//     IOTask Inputs/ControllerTags.CPX8_1[6,6] <-> Module 7 (CPX-AP-I-8DI-M8-3P)/Inputs/Input 5
//     IOTask Inputs/ControllerTags.CPX8_1[6,7] <-> Module 7 (CPX-AP-I-8DI-M8-3P)/Inputs/Input 6
//     IOTask Inputs/ControllerTags.CPX8_1[6,8] <-> Module 7 (CPX-AP-I-8DI-M8-3P)/Inputs/Input 7
//     IOTask Inputs/ControllerTags.CPX8_1[7,1] <-> Module 8 (CPX-AP-I-8DI-M8-3P)/Inputs/Input 0
//     IOTask Inputs/ControllerTags.CPX8_1[7,2] <-> Module 8 (CPX-AP-I-8DI-M8-3P)/Inputs/Input 1
//     IOTask Inputs/ControllerTags.CPX8_1[7,3] <-> Module 8 (CPX-AP-I-8DI-M8-3P)/Inputs/Input 2
//     IOTask Inputs/ControllerTags.CPX8_1[7,4] <-> Module 8 (CPX-AP-I-8DI-M8-3P)/Inputs/Input 3
//     IOTask Inputs/ControllerTags.CPX8_1[7,5] <-> Module 8 (CPX-AP-I-8DI-M8-3P)/Inputs/Input 4
//     IOTask Inputs/ControllerTags.CPX8_1[7,6] <-> Module 8 (CPX-AP-I-8DI-M8-3P)/Inputs/Input 5
//     IOTask Inputs/ControllerTags.CPX8_1[7,7] <-> Module 8 (CPX-AP-I-8DI-M8-3P)/Inputs/Input 6
//     IOTask Inputs/ControllerTags.CPX8_1[7,8] <-> Module 8 (CPX-AP-I-8DI-M8-3P)/Inputs/Input 7
//   PLC1/PLC1 Instance <-> Device 1 (EtherCAT)/Term 1 (EK1200)/Term 17 (EK1122)/Drive PA14401 (ASDA-A2-E CoE Drive)
//     PlcTask1 Inputs/ControllerTags.arErrorCodeDrive[44] <-> 1st Transmit PDO Mapping/Error code
//   PLC1/PLC1 Instance <-> Device 1 (EtherCAT)/Term 1 (EK1200)/Term 17 (EK1122)/Drive PA14501 (ASDA-A2-E CoE Drive)
//     PlcTask1 Inputs/ControllerTags.arErrorCodeDrive[45] <-> 1st Transmit PDO Mapping/Error code
//   PLC1/PLC1 Instance <-> Device 1 (EtherCAT)/Term 1 (EK1200)/Term 17 (EK1122)/Drive PA14601 (ASDA-A2-E CoE Drive)
//     PlcTask1 Inputs/ControllerTags.arErrorCodeDrive[46] <-> 1st TxPDO Mapping/Error code
//   PLC1/PLC1 Instance <-> Device 1 (EtherCAT)/Term 1 (EK1200)/Term 17 (EK1122)/Drive PA14701 (ASDA-A2-E CoE Drive)
//     PlcTask1 Inputs/ControllerTags.arErrorCodeDrive[47] <-> 1st Transmit PDO Mapping/Error code
//   PLC1/PLC1 Instance <-> Device 1 (EtherCAT)/Term 1 (EK1200)/Term 17 (EK1122)/WPI_1(WPI_EtherCAt_32Bits)
//     IOTask Outputs/ControllerTags.WPI_1[1,1] <-> DO Outputs/DataOutBit 1
//     IOTask Outputs/ControllerTags.WPI_1[1,2] <-> DO Outputs/DataOutBit  2
//     IOTask Outputs/ControllerTags.WPI_1[1,3] <-> DO Outputs/DataOutBit  3
//     IOTask Outputs/ControllerTags.WPI_1[1,4] <-> DO Outputs/DataOutBit  4
//     IOTask Outputs/ControllerTags.WPI_1[1,5] <-> DO Outputs/DataOutBit  5
//     IOTask Outputs/ControllerTags.WPI_1[1,6] <-> DO Outputs/DataOutBit  6
//     IOTask Outputs/ControllerTags.WPI_1[1,7] <-> DO Outputs/DataOutBit  7
//     IOTask Outputs/ControllerTags.WPI_1[1,8] <-> DO Outputs/DataOutBit  8
//     IOTask Outputs/ControllerTags.WPI_1[2,1] <-> DO Outputs/DataOutBit  9
//     IOTask Outputs/ControllerTags.WPI_1[2,2] <-> DO Outputs/DataOutBit  10
//     IOTask Outputs/ControllerTags.WPI_1[2,3] <-> DO Outputs/DataOutBit  11
//     IOTask Outputs/ControllerTags.WPI_1[2,4] <-> DO Outputs/DataOutBit  12
//     IOTask Outputs/ControllerTags.WPI_1[2,5] <-> DO Outputs/DataOutBit  13
//     IOTask Outputs/ControllerTags.WPI_1[2,6] <-> DO Outputs/DataOutBit  14
//     IOTask Outputs/ControllerTags.WPI_1[2,7] <-> DO Outputs/DataOutBit  15
//     IOTask Outputs/ControllerTags.WPI_1[2,8] <-> DO Outputs/DataOutBit  16
//     IOTask Outputs/ControllerTags.WPI_1[3,1] <-> DO Outputs/DataOutBit  17
//     IOTask Outputs/ControllerTags.WPI_1[3,2] <-> DO Outputs/DataOutBit  18
//     IOTask Outputs/ControllerTags.WPI_1[3,3] <-> DO Outputs/DataOutBit  19
//     IOTask Outputs/ControllerTags.WPI_1[3,4] <-> DO Outputs/DataOutBit  20
//     IOTask Outputs/ControllerTags.WPI_1[3,5] <-> DO Outputs/DataOutBit  21
//     IOTask Outputs/ControllerTags.WPI_1[3,6] <-> DO Outputs/DataOutBit  22
//     IOTask Outputs/ControllerTags.WPI_1[3,7] <-> DO Outputs/DataOutBit  23
//     IOTask Outputs/ControllerTags.WPI_1[3,8] <-> DO Outputs/DataOutBit  24
//     IOTask Outputs/ControllerTags.WPI_1[4,1] <-> DO Outputs/DataOutBit  25
//     IOTask Outputs/ControllerTags.WPI_1[4,2] <-> DO Outputs/DataOutBit  26
//     IOTask Outputs/ControllerTags.WPI_1[4,3] <-> DO Outputs/DataOutBit  27
//     IOTask Outputs/ControllerTags.WPI_1[4,4] <-> DO Outputs/DataOutBit  28
//     IOTask Outputs/ControllerTags.WPI_1[4,5] <-> DO Outputs/DataOutBit  29
//     IOTask Outputs/ControllerTags.WPI_1[4,6] <-> DO Outputs/DataOutBit  30
//     IOTask Outputs/ControllerTags.WPI_1[4,7] <-> DO Outputs/DataOutBit  31
//     IOTask Outputs/ControllerTags.WPI_1[4,8] <-> DO Outputs/DataOutBit  32
//   PLC1/PLC1 Instance <-> Device 1 (EtherCAT)/Term 1 (EK1200)/Term 17 (EK1122)/WPI_2(WPI_EtherCAt_32Bits)
//     IOTask Outputs/ControllerTags.WPI_2[1,1] <-> DO Outputs/DataOutBit 1
//     IOTask Outputs/ControllerTags.WPI_2[1,2] <-> DO Outputs/DataOutBit  2
//     IOTask Outputs/ControllerTags.WPI_2[1,3] <-> DO Outputs/DataOutBit  3
//     IOTask Outputs/ControllerTags.WPI_2[1,4] <-> DO Outputs/DataOutBit  4
//     IOTask Outputs/ControllerTags.WPI_2[1,5] <-> DO Outputs/DataOutBit  5
//     IOTask Outputs/ControllerTags.WPI_2[1,6] <-> DO Outputs/DataOutBit  6
//     IOTask Outputs/ControllerTags.WPI_2[1,7] <-> DO Outputs/DataOutBit  7
//     IOTask Outputs/ControllerTags.WPI_2[1,8] <-> DO Outputs/DataOutBit  8
//     IOTask Outputs/ControllerTags.WPI_2[2,1] <-> DO Outputs/DataOutBit  9
//     IOTask Outputs/ControllerTags.WPI_2[2,2] <-> DO Outputs/DataOutBit  10
//     IOTask Outputs/ControllerTags.WPI_2[2,3] <-> DO Outputs/DataOutBit  11
//     IOTask Outputs/ControllerTags.WPI_2[2,4] <-> DO Outputs/DataOutBit  12
//     IOTask Outputs/ControllerTags.WPI_2[2,5] <-> DO Outputs/DataOutBit  13
//     IOTask Outputs/ControllerTags.WPI_2[2,6] <-> DO Outputs/DataOutBit  14
//     IOTask Outputs/ControllerTags.WPI_2[2,7] <-> DO Outputs/DataOutBit  15
//     IOTask Outputs/ControllerTags.WPI_2[2,8] <-> DO Outputs/DataOutBit  16
//     IOTask Outputs/ControllerTags.WPI_2[3,1] <-> DO Outputs/DataOutBit  17
//     IOTask Outputs/ControllerTags.WPI_2[3,2] <-> DO Outputs/DataOutBit  18
//     IOTask Outputs/ControllerTags.WPI_2[3,3] <-> DO Outputs/DataOutBit  19
//     IOTask Outputs/ControllerTags.WPI_2[3,4] <-> DO Outputs/DataOutBit  20
//     IOTask Outputs/ControllerTags.WPI_2[3,5] <-> DO Outputs/DataOutBit  21
//     IOTask Outputs/ControllerTags.WPI_2[3,6] <-> DO Outputs/DataOutBit  22
//     IOTask Outputs/ControllerTags.WPI_2[3,7] <-> DO Outputs/DataOutBit  23
//     IOTask Outputs/ControllerTags.WPI_2[3,8] <-> DO Outputs/DataOutBit  24
//     IOTask Outputs/ControllerTags.WPI_2[4,1] <-> DO Outputs/DataOutBit  25
//     IOTask Outputs/ControllerTags.WPI_2[4,2] <-> DO Outputs/DataOutBit  26
//     IOTask Outputs/ControllerTags.WPI_2[4,3] <-> DO Outputs/DataOutBit  27
//     IOTask Outputs/ControllerTags.WPI_2[4,4] <-> DO Outputs/DataOutBit  28
//     IOTask Outputs/ControllerTags.WPI_2[4,5] <-> DO Outputs/DataOutBit  29
//     IOTask Outputs/ControllerTags.WPI_2[4,6] <-> DO Outputs/DataOutBit  30
//     IOTask Outputs/ControllerTags.WPI_2[4,7] <-> DO Outputs/DataOutBit  31
//     IOTask Outputs/ControllerTags.WPI_2[4,8] <-> DO Outputs/DataOutBit  32
//   PLC1/PLC1 Instance <-> Device 1 (EtherCAT)/Term 1 (EK1200)/Term 2 (EL1008)
//     IOTask Inputs/ControllerTags.EL1008[33,{1..8}] <-> Channel {1..8}/Input  (8 links)
//   PLC1/PLC1 Instance <-> Device 1 (EtherCAT)/Term 1 (EK1200)/Term 3 (EL1008)
//     IOTask Inputs/ControllerTags.EL1008[34,{1..8}] <-> Channel {1..8}/Input  (8 links)
//   PLC1/PLC1 Instance <-> Device 1 (EtherCAT)/Term 1 (EK1200)/Term 4 (EL1008)
//     IOTask Inputs/ControllerTags.EL1008[35,{1..8}] <-> Channel {1..8}/Input  (8 links)
//   PLC1/PLC1 Instance <-> Device 1 (EtherCAT)/Term 1 (EK1200)/Term 5 (EL1008)
//     IOTask Inputs/ControllerTags.EL1008[36,{1..8}] <-> Channel {1..8}/Input  (8 links)
//   PLC1/PLC1 Instance <-> Device 1 (EtherCAT)/Term 1 (EK1200)/Term 6 (EL1008)
//     IOTask Inputs/ControllerTags.EL1008[37,{1..8}] <-> Channel {1..8}/Input  (8 links)
//   PLC1/PLC1 Instance <-> Device 1 (EtherCAT)/Term 1 (EK1200)/Term 7 (EL2008)
//     IOTask Outputs/ControllerTags.EL2008[29,{1..8}] <-> Channel {1..8}/Output  (8 links)
//   PLC1/PLC1 Instance <-> Device 1 (EtherCAT)/Term 1 (EK1200)/Term 8 (EL2008)
//     IOTask Outputs/ControllerTags.EL2008[30,{1..8}] <-> Channel {1..8}/Output  (8 links)
//   PLC1/PLC1 Instance <-> Device 1 (EtherCAT)/Term 1 (EK1200)/Term 9 (EL2008)
//     IOTask Outputs/ControllerTags.EL2008[31,{1..8}] <-> Channel {1..8}/Output  (8 links)
//   PLC1/PLC1 Instance <-> Device 4 (EtherCAT)
//     CommunicationTask Inputs/EtherCatStates.Device2_nEcMasterDeviceId <-> InfoData/DevId
//     CommunicationTask Inputs/EtherCatStates.Device2_netID <-> InfoData/AmsNetId
//   PLC1/PLC1 Instance <-> Device 4 (EtherCAT)/Drive PA10101 (ASDA-A2-E CoE Drive)
//     PlcTask1 Inputs/ControllerTags.arErrorCodeDrive[1] <-> 1st TxPDO Mapping/Error code
//   PLC1/PLC1 Instance <-> Device 4 (EtherCAT)/Drive PA10201 (ASDA-A2-E CoE Drive)
//     PlcTask1 Inputs/ControllerTags.arErrorCodeDrive[2] <-> 1st TxPDO Mapping/Error code
//   PLC1/PLC1 Instance <-> Device 4 (EtherCAT)/Drive PA10301 (ASDA-A2-E CoE Drive)
//     PlcTask1 Inputs/ControllerTags.arErrorCodeDrive[3] <-> 1st TxPDO Mapping/Error code
//   PLC1/PLC1 Instance <-> Device 4 (EtherCAT)/Drive PA10401 (ASDA-A2-E CoE Drive)
//     PlcTask1 Inputs/ControllerTags.arErrorCodeDrive[4] <-> 1st TxPDO Mapping/Error code
//   PLC1/PLC1 Instance <-> Device 4 (EtherCAT)/Drive PA10501 (ASDA-A2-E CoE Drive)
//     PlcTask1 Inputs/ControllerTags.arErrorCodeDrive[5] <-> 1st TxPDO Mapping/Error code
//   PLC1/PLC1 Instance <-> Device 4 (EtherCAT)/Drive PA10601 (ASDA-A2-E CoE Drive)
//     PlcTask1 Inputs/ControllerTags.arErrorCodeDrive[6] <-> 1st TxPDO Mapping/Error code
//   PLC1/PLC1 Instance <-> Device 4 (EtherCAT)/Drive PA10701 (ASDA-A2-E CoE Drive)
//     PlcTask1 Inputs/ControllerTags.arErrorCodeDrive[7] <-> 1st TxPDO Mapping/Error code
//   PLC1/PLC1 Instance <-> Device 4 (EtherCAT)/Drive PA10801 (ASDA-A2-E CoE Drive)
//     PlcTask1 Inputs/ControllerTags.arErrorCodeDrive[8] <-> 1st TxPDO Mapping/Error code
//   PLC1/PLC1 Instance <-> Device 4 (EtherCAT)/Drive PA10901 (ASDA-A2-E CoE Drive)
//     PlcTask1 Inputs/ControllerTags.arErrorCodeDrive[9] <-> 1st TxPDO Mapping/Error code
//   PLC1/PLC1 Instance <-> Device 4 (EtherCAT)/Drive PA11001 (ASDA-A2-E CoE Drive)
//     PlcTask1 Inputs/ControllerTags.arErrorCodeDrive[10] <-> 1st TxPDO Mapping/Error code
//   PLC1/PLC1 Instance <-> Device 4 (EtherCAT)/Drive PA11101 (ASDA-A2-E CoE Drive)
//     PlcTask1 Inputs/ControllerTags.arErrorCodeDrive[11] <-> 1st TxPDO Mapping/Error code
//   PLC1/PLC1 Instance <-> Device 4 (EtherCAT)/Drive PA11201 (ASDA-A2-E CoE Drive)
//     PlcTask1 Inputs/ControllerTags.arErrorCodeDrive[12] <-> 1st TxPDO Mapping/Error code
//   PLC1/PLC1 Instance <-> Device 4 (EtherCAT)/Drive PA11301 (ASDA-A2-E CoE Drive)
//     PlcTask1 Inputs/ControllerTags.arErrorCodeDrive[13] <-> 1st TxPDO Mapping/Error code
//   PLC1/PLC1 Instance <-> Device 4 (EtherCAT)/Drive PA11401 (ASDA-A2-E CoE Drive)
//     PlcTask1 Inputs/ControllerTags.arErrorCodeDrive[14] <-> 1st TxPDO Mapping/Error code
//   PLC1/PLC1 Instance <-> Device 4 (EtherCAT)/Drive PA11501 (ASDA-A2-E CoE Drive)
//     PlcTask1 Inputs/ControllerTags.arErrorCodeDrive[15] <-> 1st TxPDO Mapping/Error code
//   PLC1/PLC1 Instance <-> Device 4 (EtherCAT)/Drive PA11601 (ASDA-A2-E CoE Drive)
//     PlcTask1 Inputs/ControllerTags.arErrorCodeDrive[16] <-> 1st TxPDO Mapping/Error code
//   PLC1/PLC1 Instance <-> Device 4 (EtherCAT)/Drive PA11701 (ASDA-A2-E CoE Drive)
//     PlcTask1 Inputs/ControllerTags.arErrorCodeDrive[17] <-> 1st TxPDO Mapping/Error code
//   PLC1/PLC1 Instance <-> Device 4 (EtherCAT)/Drive PA11801 (ASDA-A2-E CoE Drive)
//     PlcTask1 Inputs/ControllerTags.arErrorCodeDrive[18] <-> 1st TxPDO Mapping/Error code
//   PLC1/PLC1 Instance <-> Device 4 (EtherCAT)/Drive PA11901 (ASDA-A2-E CoE Drive)
//     PlcTask1 Inputs/ControllerTags.arErrorCodeDrive[19] <-> 1st TxPDO Mapping/Error code
//   PLC1/PLC1 Instance <-> Device 4 (EtherCAT)/Drive PA12001 (ASDA-A2-E CoE Drive)
//     PlcTask1 Inputs/ControllerTags.arErrorCodeDrive[20] <-> 1st TxPDO Mapping/Error code
//   PLC1/PLC1 Instance <-> Device 4 (EtherCAT)/Drive PA12101 (ASDA-A2-E CoE Drive)
//     PlcTask1 Inputs/ControllerTags.arErrorCodeDrive[41] <-> 1st TxPDO Mapping/Error code
//   PLC1/PLC1 Instance <-> Device 4 (EtherCAT)/Drive PA12201 (ASDA-A2-E CoE Drive)
//     PlcTask1 Inputs/ControllerTags.arErrorCodeDrive[21] <-> 1st TxPDO Mapping/Error code
//   PLC1/PLC1 Instance <-> Device 4 (EtherCAT)/Drive PA12301 (ASDA-A2-E CoE Drive)
//     PlcTask1 Inputs/ControllerTags.arErrorCodeDrive[22] <-> 1st TxPDO Mapping/Error code
//   PLC1/PLC1 Instance <-> Device 4 (EtherCAT)/Drive PA12401 (ASDA-A2-E CoE Drive)
//     PlcTask1 Inputs/ControllerTags.arErrorCodeDrive[23] <-> 1st TxPDO Mapping/Error code
//   PLC1/PLC1 Instance <-> Device 4 (EtherCAT)/Drive PA12501 (ASDA-A2-E CoE Drive)
//     PlcTask1 Inputs/ControllerTags.arErrorCodeDrive[24] <-> 1st TxPDO Mapping/Error code
//   PLC1/PLC1 Instance <-> Device 4 (EtherCAT)/Drive PA12601 (ASDA-A2-E CoE Drive)
//     PlcTask1 Inputs/ControllerTags.arErrorCodeDrive[25] <-> 1st TxPDO Mapping/Error code
//   PLC1/PLC1 Instance <-> Device 4 (EtherCAT)/Drive PA12701 (ASDA-A2-E CoE Drive)
//     PlcTask1 Inputs/ControllerTags.arErrorCodeDrive[26] <-> 1st TxPDO Mapping/Error code
//   PLC1/PLC1 Instance <-> Device 4 (EtherCAT)/Drive PA12801 (ASDA-A2-E CoE Drive)
//     PlcTask1 Inputs/ControllerTags.arErrorCodeDrive[27] <-> 1st TxPDO Mapping/Error code
//   PLC1/PLC1 Instance <-> Device 4 (EtherCAT)/Drive PA12901 (ASDA-A2-E CoE Drive)
//     PlcTask1 Inputs/ControllerTags.arErrorCodeDrive[28] <-> 1st TxPDO Mapping/Error code
//   PLC1/PLC1 Instance <-> Device 4 (EtherCAT)/Drive PA13001 (ASDA-A2-E CoE Drive)
//     PlcTask1 Inputs/ControllerTags.arErrorCodeDrive[29] <-> 1st TxPDO Mapping/Error code
//   PLC1/PLC1 Instance <-> Device 4 (EtherCAT)/Drive PA13101 (ASDA-A2-E CoE Drive)
//     PlcTask1 Inputs/ControllerTags.arErrorCodeDrive[30] <-> 1st TxPDO Mapping/Error code
//   PLC1/PLC1 Instance <-> Device 4 (EtherCAT)/Drive PA13201 (ASDA-A2-E CoE Drive)
//     PlcTask1 Inputs/ControllerTags.arErrorCodeDrive[42] <-> 1st TxPDO Mapping/Error code
//   PLC1/PLC1 Instance <-> Device 4 (EtherCAT)/Drive PA13301 (ASDA-A2-E CoE Drive)
//     PlcTask1 Inputs/ControllerTags.arErrorCodeDrive[31] <-> 1st Transmit PDO Mapping/Error code
//   PLC1/PLC1 Instance <-> Device 4 (EtherCAT)/Drive PA13401 (ASDA-A2-E CoE Drive)
//     PlcTask1 Inputs/ControllerTags.arErrorCodeDrive[32] <-> 1st Transmit PDO Mapping/Error code
//   PLC1/PLC1 Instance <-> Device 4 (EtherCAT)/Drive PA13501 (ASDA-A2-E CoE Drive)
//     PlcTask1 Inputs/ControllerTags.arErrorCodeDrive[33] <-> 1st Transmit PDO Mapping/Error code
//   PLC1/PLC1 Instance <-> Device 4 (EtherCAT)/Drive PA13601 (ASDA-A2-E CoE Drive)
//     PlcTask1 Inputs/ControllerTags.arErrorCodeDrive[34] <-> 1st TxPDO Mapping/Error code
//   PLC1/PLC1 Instance <-> Device 4 (EtherCAT)/Drive PA13701 (ASDA-A2-E CoE Drive)
//     PlcTask1 Inputs/ControllerTags.arErrorCodeDrive[35] <-> 1st TxPDO Mapping/Error code
//   PLC1/PLC1 Instance <-> Device 4 (EtherCAT)/Drive PA13801 (ASDA-A2-E CoE Drive)
//     PlcTask1 Inputs/ControllerTags.arErrorCodeDrive[36] <-> 1st TxPDO Mapping/Error code
//   PLC1/PLC1 Instance <-> Device 4 (EtherCAT)/Drive PA13901 (ASDA-A2-E CoE Drive)
//     PlcTask1 Inputs/ControllerTags.arErrorCodeDrive[37] <-> 1st TxPDO Mapping/Error code
//   PLC1/PLC1 Instance <-> Device 4 (EtherCAT)/Drive PA14001 (ASDA-A2-E CoE Drive)
//     PlcTask1 Inputs/ControllerTags.arErrorCodeDrive[38] <-> 1st TxPDO Mapping/Error code
//   PLC1/PLC1 Instance <-> Device 4 (EtherCAT)/Drive PA14101 (ASDA-A2-E CoE Drive)
//     PlcTask1 Inputs/ControllerTags.arErrorCodeDrive[39] <-> 1st TxPDO Mapping/Error code
//   PLC1/PLC1 Instance <-> Device 4 (EtherCAT)/Drive PA14201 (ASDA-A2-E CoE Drive)
//     PlcTask1 Inputs/ControllerTags.arErrorCodeDrive[40] <-> 1st TxPDO Mapping/Error code
//   PLC1/PLC1 Instance <-> Device 4 (EtherCAT)/Drive PA14301 (ASDA-A2-E CoE Drive)
//     PlcTask1 Inputs/ControllerTags.arErrorCodeDrive[43] <-> 1st TxPDO Mapping/Error code
//   PLC1/PLC1 Instance <-> Device 4 (EtherCAT)/Term CIM32101 (EK1100)/Term 110 (EL1008)
//     IOTask Inputs/ControllerTags.EL1008[1,{1..8}] <-> Channel {1..8}/Input  (8 links)
//   PLC1/PLC1 Instance <-> Device 4 (EtherCAT)/Term CIM32101 (EK1100)/Term 111 (EL1008)
//     IOTask Inputs/ControllerTags.EL1008[2,{1..8}] <-> Channel {1..8}/Input  (8 links)
//   PLC1/PLC1 Instance <-> Device 4 (EtherCAT)/Term CIM32101 (EK1100)/Term 112 (EL1008)
//     IOTask Inputs/ControllerTags.EL1008[3,{1..8}] <-> Channel {1..8}/Input  (8 links)
//   PLC1/PLC1 Instance <-> Device 4 (EtherCAT)/Term CIM32101 (EK1100)/Term 113 (EL1008)
//     IOTask Inputs/ControllerTags.EL1008[4,{1..8}] <-> Channel {1..8}/Input  (8 links)
//   PLC1/PLC1 Instance <-> Device 4 (EtherCAT)/Term CIM32101 (EK1100)/Term 114 (EL1008)
//     IOTask Inputs/ControllerTags.EL1008[5,{1..8}] <-> Channel {1..8}/Input  (8 links)
//   PLC1/PLC1 Instance <-> Device 4 (EtherCAT)/Term CIM32101 (EK1100)/Term 115 (EL1008)
//     IOTask Inputs/ControllerTags.EL1008[6,{1..8}] <-> Channel {1..8}/Input  (8 links)
//   PLC1/PLC1 Instance <-> Device 4 (EtherCAT)/Term CIM32101 (EK1100)/Term 116 (EL1008)
//     IOTask Inputs/ControllerTags.EL1008[7,{1..8}] <-> Channel {1..8}/Input  (8 links)
//   PLC1/PLC1 Instance <-> Device 4 (EtherCAT)/Term CIM32101 (EK1100)/Term 117 (EL1008)
//     IOTask Inputs/ControllerTags.EL1008[29,{1..8}] <-> Channel {1..8}/Input  (8 links)
//   PLC1/PLC1 Instance <-> Device 4 (EtherCAT)/Term CIM32101 (EK1100)/Term 118 (EL2008)
//     IOTask Outputs/ControllerTags.EL2008[1,{1..8}] <-> Channel {1..8}/Output  (8 links)
//   PLC1/PLC1 Instance <-> Device 4 (EtherCAT)/Term CIM32101 (EK1100)/Term 119 (EL2008)
//     IOTask Outputs/ControllerTags.EL2008[2,{1..8}] <-> Channel {1..8}/Output  (8 links)
//   PLC1/PLC1 Instance <-> Device 4 (EtherCAT)/Term CIM32101 (EK1100)/Term 120 (EL2008)
//     IOTask Outputs/ControllerTags.EL2008[3,{1..8}] <-> Channel {1..8}/Output  (8 links)
//   PLC1/PLC1 Instance <-> Device 4 (EtherCAT)/Term CIM32101 (EK1100)/Term 121 (EL2008)
//     IOTask Outputs/ControllerTags.EL2008[4,{1..8}] <-> Channel {1..8}/Output  (8 links)
//   PLC1/PLC1 Instance <-> Device 4 (EtherCAT)/Term CIM32101 (EK1100)/Term 122 (EL2008)
//     IOTask Outputs/ControllerTags.EL2008[5,{1..8}] <-> Channel {1..8}/Output  (8 links)
//   PLC1/PLC1 Instance <-> Device 4 (EtherCAT)/Term CIM32101 (EK1100)/Term 123 (EL2008)
//     IOTask Outputs/ControllerTags.EL2008[6,{1..8}] <-> Channel {1..8}/Output  (8 links)
//   PLC1/PLC1 Instance <-> Device 4 (EtherCAT)/Term CIM32101 (EK1100)/Term 124 (EL2008)
//     IOTask Outputs/ControllerTags.EL2008[7,{1..8}] <-> Channel {1..8}/Output  (8 links)
//   PLC1/PLC1 Instance <-> Device 4 (EtherCAT)/Term CIM33701 (EK1100)/Term 83 (EL1008)
//     IOTask Inputs/ControllerTags.EL1008[8,{1..8}] <-> Channel {1..8}/Input  (8 links)
//   PLC1/PLC1 Instance <-> Device 4 (EtherCAT)/Term CIM33701 (EK1100)/Term 84 (EL1008)
//     IOTask Inputs/ControllerTags.EL1008[9,{1..8}] <-> Channel {1..8}/Input  (8 links)
//   PLC1/PLC1 Instance <-> Device 4 (EtherCAT)/Term CIM33701 (EK1100)/Term 85 (EL1008)
//     IOTask Inputs/ControllerTags.EL1008[10,{1..8}] <-> Channel {1..8}/Input  (8 links)
//   PLC1/PLC1 Instance <-> Device 4 (EtherCAT)/Term CIM33701 (EK1100)/Term 86 (EL1008)
//     IOTask Inputs/ControllerTags.EL1008[11,{1..8}] <-> Channel {1..8}/Input  (8 links)
//   PLC1/PLC1 Instance <-> Device 4 (EtherCAT)/Term CIM33701 (EK1100)/Term 87 (EL1008)
//     IOTask Inputs/ControllerTags.EL1008[12,{1..8}] <-> Channel {1..8}/Input  (8 links)
//   PLC1/PLC1 Instance <-> Device 4 (EtherCAT)/Term CIM33701 (EK1100)/Term 88 (EL1008)
//     IOTask Inputs/ControllerTags.EL1008[13,{1..8}] <-> Channel {1..8}/Input  (8 links)
//   PLC1/PLC1 Instance <-> Device 4 (EtherCAT)/Term CIM33701 (EK1100)/Term 89 (EL1008)
//     IOTask Inputs/ControllerTags.EL1008[14,{1..8}] <-> Channel {1..8}/Input  (8 links)
//   PLC1/PLC1 Instance <-> Device 4 (EtherCAT)/Term CIM33701 (EK1100)/Term 90 (EL1008)
//     IOTask Inputs/ControllerTags.EL1008[30,{1..8}] <-> Channel {1..8}/Input  (8 links)
//   PLC1/PLC1 Instance <-> Device 4 (EtherCAT)/Term CIM33701 (EK1100)/Term 91 (EL2008)
//     IOTask Outputs/ControllerTags.EL2008[8,{1..8}] <-> Channel {1..8}/Output  (8 links)
//   PLC1/PLC1 Instance <-> Device 4 (EtherCAT)/Term CIM33701 (EK1100)/Term 92 (EL2008)
//     IOTask Outputs/ControllerTags.EL2008[9,{1..8}] <-> Channel {1..8}/Output  (8 links)
//   PLC1/PLC1 Instance <-> Device 4 (EtherCAT)/Term CIM33701 (EK1100)/Term 93 (EL2008)
//     IOTask Outputs/ControllerTags.EL2008[10,{1..8}] <-> Channel {1..8}/Output  (8 links)
//   PLC1/PLC1 Instance <-> Device 4 (EtherCAT)/Term CIM33701 (EK1100)/Term 94 (EL2008)
//     IOTask Outputs/ControllerTags.EL2008[11,{1..8}] <-> Channel {1..8}/Output  (8 links)
//   PLC1/PLC1 Instance <-> Device 4 (EtherCAT)/Term CIM33701 (EK1100)/Term 95 (EL2008)
//     IOTask Outputs/ControllerTags.EL2008[12,{1..8}] <-> Channel {1..8}/Output  (8 links)
//   PLC1/PLC1 Instance <-> Device 4 (EtherCAT)/Term CIM33701 (EK1100)/Term 96 (EL2008)
//     IOTask Outputs/ControllerTags.EL2008[13,{1..8}] <-> Channel {1..8}/Output  (8 links)
//   PLC1/PLC1 Instance <-> Device 4 (EtherCAT)/Term CIM33701 (EK1100)/Term 97 (EL2008)
//     IOTask Outputs/ControllerTags.EL2008[14,{1..8}] <-> Channel {1..8}/Output  (8 links)
//   PLC1/PLC1 Instance <-> Device 4 (EtherCAT)/Term CIM35301 (EK1100)/Term 56 (EL1008)
//     IOTask Inputs/ControllerTags.EL1008[15,{1..8}] <-> Channel {1..8}/Input  (8 links)
//   PLC1/PLC1 Instance <-> Device 4 (EtherCAT)/Term CIM35301 (EK1100)/Term 57 (EL1008)
//     IOTask Inputs/ControllerTags.EL1008[16,{1..8}] <-> Channel {1..8}/Input  (8 links)
//   PLC1/PLC1 Instance <-> Device 4 (EtherCAT)/Term CIM35301 (EK1100)/Term 58 (EL1008)
//     IOTask Inputs/ControllerTags.EL1008[17,{1..8}] <-> Channel {1..8}/Input  (8 links)
//   PLC1/PLC1 Instance <-> Device 4 (EtherCAT)/Term CIM35301 (EK1100)/Term 59 (EL1008)
//     IOTask Inputs/ControllerTags.EL1008[18,{1..8}] <-> Channel {1..8}/Input  (8 links)
//   PLC1/PLC1 Instance <-> Device 4 (EtherCAT)/Term CIM35301 (EK1100)/Term 60 (EL1008)
//     IOTask Inputs/ControllerTags.EL1008[19,{1..8}] <-> Channel {1..8}/Input  (8 links)
//   PLC1/PLC1 Instance <-> Device 4 (EtherCAT)/Term CIM35301 (EK1100)/Term 61 (EL1008)
//     IOTask Inputs/ControllerTags.EL1008[20,{1..8}] <-> Channel {1..8}/Input  (8 links)
//   PLC1/PLC1 Instance <-> Device 4 (EtherCAT)/Term CIM35301 (EK1100)/Term 62 (EL1008)
//     IOTask Inputs/ControllerTags.EL1008[21,{1..8}] <-> Channel {1..8}/Input  (8 links)
//   PLC1/PLC1 Instance <-> Device 4 (EtherCAT)/Term CIM35301 (EK1100)/Term 63 (EL1008)
//     IOTask Inputs/ControllerTags.EL1008[31,{1..8}] <-> Channel {1..8}/Input  (8 links)
//   PLC1/PLC1 Instance <-> Device 4 (EtherCAT)/Term CIM35301 (EK1100)/Term 64 (EL2008)
//     IOTask Outputs/ControllerTags.EL2008[15,{1..8}] <-> Channel {1..8}/Output  (8 links)
//   PLC1/PLC1 Instance <-> Device 4 (EtherCAT)/Term CIM35301 (EK1100)/Term 65 (EL2008)
//     IOTask Outputs/ControllerTags.EL2008[16,{1..8}] <-> Channel {1..8}/Output  (8 links)
//   PLC1/PLC1 Instance <-> Device 4 (EtherCAT)/Term CIM35301 (EK1100)/Term 66 (EL2008)
//     IOTask Outputs/ControllerTags.EL2008[17,{1..8}] <-> Channel {1..8}/Output  (8 links)
//   PLC1/PLC1 Instance <-> Device 4 (EtherCAT)/Term CIM35301 (EK1100)/Term 67 (EL2008)
//     IOTask Outputs/ControllerTags.EL2008[18,{1..8}] <-> Channel {1..8}/Output  (8 links)
//   PLC1/PLC1 Instance <-> Device 4 (EtherCAT)/Term CIM35301 (EK1100)/Term 68 (EL2008)
//     IOTask Outputs/ControllerTags.EL2008[19,{1..8}] <-> Channel {1..8}/Output  (8 links)
//   PLC1/PLC1 Instance <-> Device 4 (EtherCAT)/Term CIM35301 (EK1100)/Term 69 (EL2008)
//     IOTask Outputs/ControllerTags.EL2008[20,{1..8}] <-> Channel {1..8}/Output  (8 links)
//   PLC1/PLC1 Instance <-> Device 4 (EtherCAT)/Term CIM35301 (EK1100)/Term 70 (EL2008)
//     IOTask Outputs/ControllerTags.EL2008[21,{1..8}] <-> Channel {1..8}/Output  (8 links)
//   PLC1/PLC1 Instance <-> Device 4 (EtherCAT)/Term CIM36901 (EK1100)/Term 29 (EL1008)
//     IOTask Inputs/ControllerTags.EL1008[22,{1..8}] <-> Channel {1..8}/Input  (8 links)
//   PLC1/PLC1 Instance <-> Device 4 (EtherCAT)/Term CIM36901 (EK1100)/Term 30 (EL1008)
//     IOTask Inputs/ControllerTags.EL1008[23,{1..8}] <-> Channel {1..8}/Input  (8 links)
//   PLC1/PLC1 Instance <-> Device 4 (EtherCAT)/Term CIM36901 (EK1100)/Term 31 (EL1008)
//     IOTask Inputs/ControllerTags.EL1008[24,{1..8}] <-> Channel {1..8}/Input  (8 links)
//   PLC1/PLC1 Instance <-> Device 4 (EtherCAT)/Term CIM36901 (EK1100)/Term 32 (EL1008)
//     IOTask Inputs/ControllerTags.EL1008[25,{1..8}] <-> Channel {1..8}/Input  (8 links)
//   PLC1/PLC1 Instance <-> Device 4 (EtherCAT)/Term CIM36901 (EK1100)/Term 33 (EL1008)
//     IOTask Inputs/ControllerTags.EL1008[26,{1..8}] <-> Channel {1..8}/Input  (8 links)
//   PLC1/PLC1 Instance <-> Device 4 (EtherCAT)/Term CIM36901 (EK1100)/Term 34 (EL1008)
//     IOTask Inputs/ControllerTags.EL1008[27,{1..8}] <-> Channel {1..8}/Input  (8 links)
//   PLC1/PLC1 Instance <-> Device 4 (EtherCAT)/Term CIM36901 (EK1100)/Term 35 (EL1008)
//     IOTask Inputs/ControllerTags.EL1008[28,{1..8}] <-> Channel {1..8}/Input  (8 links)
//   PLC1/PLC1 Instance <-> Device 4 (EtherCAT)/Term CIM36901 (EK1100)/Term 36 (EL1008)
//     IOTask Inputs/ControllerTags.EL1008[32,{1..8}] <-> Channel {1..8}/Input  (8 links)
//   PLC1/PLC1 Instance <-> Device 4 (EtherCAT)/Term CIM36901 (EK1100)/Term 37 (EL2008)
//     IOTask Outputs/ControllerTags.EL2008[22,{1..8}] <-> Channel {1..8}/Output  (8 links)
//   PLC1/PLC1 Instance <-> Device 4 (EtherCAT)/Term CIM36901 (EK1100)/Term 38 (EL2008)
//     IOTask Outputs/ControllerTags.EL2008[23,{1..8}] <-> Channel {1..8}/Output  (8 links)
//   PLC1/PLC1 Instance <-> Device 4 (EtherCAT)/Term CIM36901 (EK1100)/Term 39 (EL2008)
//     IOTask Outputs/ControllerTags.EL2008[24,{1..8}] <-> Channel {1..8}/Output  (8 links)
//   PLC1/PLC1 Instance <-> Device 4 (EtherCAT)/Term CIM36901 (EK1100)/Term 40 (EL2008)
//     IOTask Outputs/ControllerTags.EL2008[25,{1..8}] <-> Channel {1..8}/Output  (8 links)
//   PLC1/PLC1 Instance <-> Device 4 (EtherCAT)/Term CIM36901 (EK1100)/Term 41 (EL2008)
//     IOTask Outputs/ControllerTags.EL2008[26,{1..8}] <-> Channel {1..8}/Output  (8 links)
//   PLC1/PLC1 Instance <-> Device 4 (EtherCAT)/Term CIM36901 (EK1100)/Term 42 (EL2008)
//     IOTask Outputs/ControllerTags.EL2008[27,{1..8}] <-> Channel {1..8}/Output  (8 links)
//   PLC1/PLC1 Instance <-> Device 4 (EtherCAT)/Term CIM36901 (EK1100)/Term 43 (EL2008)
//     IOTask Outputs/ControllerTags.EL2008[28,{1..8}] <-> Channel {1..8}/Output  (8 links)
//   PLC1/PLC1 Instance <-> Device 6 (NOV-DP-RAM)/Box 18 (Retain Handler)
//     CommunicationTask Retains/ControllerTags.HMI_CutNo <-> Retains/ControllerTags.HMI_CutNo_[851]
//     CommunicationTask Retains/ControllerTags.HMI_DropPosOffset <-> Retains/ControllerTags.HMI_DropPosOffset_[851]
//     CommunicationTask Retains/ControllerTags.HMI_EMSelectUN02 <-> Retains/ControllerTags.HMI_EMSelectUN02_[851]
//     CommunicationTask Retains/ControllerTags.HMI_PickNo <-> Retains/ControllerTags.HMI_PickNo_[851]
//     CommunicationTask Retains/ControllerTags.HMI_PrintMaxTime <-> Retains/ControllerTags.HMI_PrintMaxTime_[851]
//     CommunicationTask Retains/ControllerTags.HMI_PusherPos <-> Retains/ControllerTags.HMI_PusherPos_[851]
//     PlcTask1 Retains/ControllerTags.HMI_B1DropBinNo <-> Retains/ControllerTags.HMI_B1DropBinNo_[851]
//     PlcTask1 Retains/ControllerTags.HMI_B2DropBinNo <-> Retains/ControllerTags.HMI_B2DropBinNo_[851]
//     PlcTask1 Retains/ControllerTags.HMI_B3DropBinNo1 <-> Retains/ControllerTags.HMI_B3DropBinNo1_[851]
//     PlcTask1 Retains/ControllerTags.HMI_B3DropBinNo2 <-> Retains/ControllerTags.HMI_B3DropBinNo2_[851]
//     PlcTask1 Retains/ControllerTags.HMI_B3DropBinNo3 <-> Retains/ControllerTags.HMI_B3DropBinNo3_[851]
//     PlcTask1 Retains/ControllerTags.HMI_BeltAcc <-> Retains/ControllerTags.HMI_BeltAcc_[851]
//     PlcTask1 Retains/ControllerTags.HMI_BeltDec <-> Retains/ControllerTags.HMI_BeltDec_[851]
//     PlcTask1 Retains/ControllerTags.HMI_BeltVelo <-> Retains/ControllerTags.HMI_BeltVelo_[851]
//     PlcTask1 Retains/ControllerTags.HMI_Check1No <-> Retains/ControllerTags.HMI_Check1No_[851]
//     PlcTask1 Retains/ControllerTags.HMI_Check2No <-> Retains/ControllerTags.HMI_Check2No_[851]
//     PlcTask1 Retains/ControllerTags.HMI_CntCheck <-> Retains/ControllerTags.HMI_CntCheck_[851]
//     PlcTask1 Retains/ControllerTags.HMI_CntCheckTime <-> Retains/ControllerTags.HMI_CntCheckTime_[851]
//     PlcTask1 Retains/ControllerTags.HMI_CountersAcc <-> Retains/ControllerTags.HMI_CountersAcc_[851]
//     PlcTask1 Retains/ControllerTags.HMI_CountersDec <-> Retains/ControllerTags.HMI_CountersDec_[851]
//     PlcTask1 Retains/ControllerTags.HMI_CountersVelo <-> Retains/ControllerTags.HMI_CountersVelo_[851]
//     PlcTask1 Retains/ControllerTags.HMI_DropNo <-> Retains/ControllerTags.HMI_DropNo_[851]
//     PlcTask1 Retains/ControllerTags.HMI_EMSelectUN01 <-> Retains/ControllerTags.HMI_EMSelectUN01_[851]
//     PlcTask1 Retains/ControllerTags.HMI_HeatTempSet <-> Retains/ControllerTags.HMI_HeatTempSet_[851]
//     PlcTask1 Retains/ControllerTags.HMI_HomeOffsetBelt <-> Retains/ControllerTags.HMI_HomeOffsetBelt_[851]
//     PlcTask1 Retains/ControllerTags.HMI_MasterVelo <-> Retains/ControllerTags.HMI_MasterVelo_[851]
//     PlcTask1 Retains/ControllerTags.HMI_PrintNo <-> Retains/ControllerTags.HMI_PrintNo_[851]
//     PlcTask1 Retains/ControllerTags.HMI_PullerPara <-> Retains/ControllerTags.HMI_PullerPara_[851]
//     PlcTask1 Retains/ControllerTags.HMI_Seal1No <-> Retains/ControllerTags.HMI_Seal1No_[851]
//     PlcTask1 Retains/ControllerTags.HMI_Seal2No <-> Retains/ControllerTags.HMI_Seal2No_[851]
//     PlcTask1 Retains/ControllerTags.HMI_SealTime <-> Retains/ControllerTags.HMI_SealTime_[851]
//     PlcTask1 Retains/ControllerTags.HMI_SealTime2 <-> Retains/ControllerTags.HMI_SealTime2_[851]
//     PlcTask1 Retains/ControllerTags.HMI_SkipCntAlarm <-> Retains/ControllerTags.HMI_SkipCntAlarm_[851]
//     PlcTask1 Retains/ControllerTags.HMI_TransferNo <-> Retains/ControllerTags.HMI_TransferNo_[851]
//     PlcTask1 Retains/ControllerTags.HMI_arSealTime <-> Retains/ControllerTags.HMI_arSealTime_[851]
//   PLC1/PLC1 Instance <-> NC-Task 1 SAF/Axes/Belt 1
//     MotionTask Inputs/ControllerTags.arRealAxisAdmin[41].Axis.NcToPlc <-> Outputs/ToPlc
//     MotionTask Outputs/ControllerTags.arRealAxisAdmin[41].Axis.PlcToNc <-> Inputs/FromPlc
//   PLC1/PLC1 Instance <-> NC-Task 1 SAF/Axes/Belt 2
//     MotionTask Inputs/ControllerTags.arRealAxisAdmin[42].Axis.NcToPlc <-> Outputs/ToPlc
//     MotionTask Outputs/ControllerTags.arRealAxisAdmin[42].Axis.PlcToNc <-> Inputs/FromPlc
//   PLC1/PLC1 Instance <-> NC-Task 1 SAF/Axes/Belt 3
//     MotionTask Inputs/ControllerTags.arRealAxisAdmin[43].Axis.NcToPlc <-> Outputs/ToPlc
//     MotionTask Outputs/ControllerTags.arRealAxisAdmin[43].Axis.PlcToNc <-> Inputs/FromPlc
//   PLC1/PLC1 Instance <-> NC-Task 1 SAF/Axes/Belt 4
//     MotionTask Inputs/ControllerTags.arRealAxisAdmin[44].Axis.NcToPlc <-> Outputs/ToPlc
//     MotionTask Outputs/ControllerTags.arRealAxisAdmin[44].Axis.PlcToNc <-> Inputs/FromPlc
//   PLC1/PLC1 Instance <-> NC-Task 1 SAF/Axes/Belt 5
//     MotionTask Inputs/ControllerTags.arRealAxisAdmin[45].Axis.NcToPlc <-> Outputs/ToPlc
//     MotionTask Outputs/ControllerTags.arRealAxisAdmin[45].Axis.PlcToNc <-> Inputs/FromPlc
//   PLC1/PLC1 Instance <-> NC-Task 1 SAF/Axes/Belt 6
//     MotionTask Inputs/ControllerTags.arRealAxisAdmin[46].Axis.NcToPlc <-> Outputs/ToPlc
//     MotionTask Outputs/ControllerTags.arRealAxisAdmin[46].Axis.PlcToNc <-> Inputs/FromPlc
//   PLC1/PLC1 Instance <-> NC-Task 1 SAF/Axes/Belt7
//     MotionTask Inputs/ControllerTags.arRealAxisAdmin[48].Axis.NcToPlc <-> Outputs/ToPlc
//     MotionTask Outputs/ControllerTags.arRealAxisAdmin[48].Axis.PlcToNc <-> Inputs/FromPlc
//   PLC1/PLC1 Instance <-> NC-Task 1 SAF/Axes/Counter 1
//     MotionTask Inputs/ControllerTags.arRealAxisAdmin[1].Axis.NcToPlc <-> Outputs/ToPlc
//     MotionTask Outputs/ControllerTags.arRealAxisAdmin[1].Axis.PlcToNc <-> Inputs/FromPlc
//   PLC1/PLC1 Instance <-> NC-Task 1 SAF/Axes/Counter 10
//     MotionTask Inputs/ControllerTags.arRealAxisAdmin[10].Axis.NcToPlc <-> Outputs/ToPlc
//     MotionTask Outputs/ControllerTags.arRealAxisAdmin[10].Axis.PlcToNc <-> Inputs/FromPlc
//   PLC1/PLC1 Instance <-> NC-Task 1 SAF/Axes/Counter 11
//     MotionTask Inputs/ControllerTags.arRealAxisAdmin[11].Axis.NcToPlc <-> Outputs/ToPlc
//     MotionTask Outputs/ControllerTags.arRealAxisAdmin[11].Axis.PlcToNc <-> Inputs/FromPlc
//   PLC1/PLC1 Instance <-> NC-Task 1 SAF/Axes/Counter 12
//     MotionTask Inputs/ControllerTags.arRealAxisAdmin[12].Axis.NcToPlc <-> Outputs/ToPlc
//     MotionTask Outputs/ControllerTags.arRealAxisAdmin[12].Axis.PlcToNc <-> Inputs/FromPlc
//   PLC1/PLC1 Instance <-> NC-Task 1 SAF/Axes/Counter 13
//     MotionTask Inputs/ControllerTags.arRealAxisAdmin[13].Axis.NcToPlc <-> Outputs/ToPlc
//     MotionTask Outputs/ControllerTags.arRealAxisAdmin[13].Axis.PlcToNc <-> Inputs/FromPlc
//   PLC1/PLC1 Instance <-> NC-Task 1 SAF/Axes/Counter 14
//     MotionTask Inputs/ControllerTags.arRealAxisAdmin[14].Axis.NcToPlc <-> Outputs/ToPlc
//     MotionTask Outputs/ControllerTags.arRealAxisAdmin[14].Axis.PlcToNc <-> Inputs/FromPlc
//   PLC1/PLC1 Instance <-> NC-Task 1 SAF/Axes/Counter 15
//     MotionTask Inputs/ControllerTags.arRealAxisAdmin[15].Axis.NcToPlc <-> Outputs/ToPlc
//     MotionTask Outputs/ControllerTags.arRealAxisAdmin[15].Axis.PlcToNc <-> Inputs/FromPlc
//   PLC1/PLC1 Instance <-> NC-Task 1 SAF/Axes/Counter 16
//     MotionTask Inputs/ControllerTags.arRealAxisAdmin[16].Axis.NcToPlc <-> Outputs/ToPlc
//     MotionTask Outputs/ControllerTags.arRealAxisAdmin[16].Axis.PlcToNc <-> Inputs/FromPlc
//   PLC1/PLC1 Instance <-> NC-Task 1 SAF/Axes/Counter 17
//     MotionTask Inputs/ControllerTags.arRealAxisAdmin[17].Axis.NcToPlc <-> Outputs/ToPlc
//     MotionTask Outputs/ControllerTags.arRealAxisAdmin[17].Axis.PlcToNc <-> Inputs/FromPlc
//   PLC1/PLC1 Instance <-> NC-Task 1 SAF/Axes/Counter 18
//     MotionTask Inputs/ControllerTags.arRealAxisAdmin[18].Axis.NcToPlc <-> Outputs/ToPlc
//     MotionTask Outputs/ControllerTags.arRealAxisAdmin[18].Axis.PlcToNc <-> Inputs/FromPlc
//   PLC1/PLC1 Instance <-> NC-Task 1 SAF/Axes/Counter 19
//     MotionTask Inputs/ControllerTags.arRealAxisAdmin[19].Axis.NcToPlc <-> Outputs/ToPlc
//     MotionTask Outputs/ControllerTags.arRealAxisAdmin[19].Axis.PlcToNc <-> Inputs/FromPlc
//   PLC1/PLC1 Instance <-> NC-Task 1 SAF/Axes/Counter 2
//     MotionTask Inputs/ControllerTags.arRealAxisAdmin[2].Axis.NcToPlc <-> Outputs/ToPlc
//     MotionTask Outputs/ControllerTags.arRealAxisAdmin[2].Axis.PlcToNc <-> Inputs/FromPlc
//   PLC1/PLC1 Instance <-> NC-Task 1 SAF/Axes/Counter 20
//     MotionTask Inputs/ControllerTags.arRealAxisAdmin[20].Axis.NcToPlc <-> Outputs/ToPlc
//     MotionTask Outputs/ControllerTags.arRealAxisAdmin[20].Axis.PlcToNc <-> Inputs/FromPlc
//   PLC1/PLC1 Instance <-> NC-Task 1 SAF/Axes/Counter 21
//     MotionTask Inputs/ControllerTags.arRealAxisAdmin[21].Axis.NcToPlc <-> Outputs/ToPlc
//     MotionTask Outputs/ControllerTags.arRealAxisAdmin[21].Axis.PlcToNc <-> Inputs/FromPlc
//   PLC1/PLC1 Instance <-> NC-Task 1 SAF/Axes/Counter 22
//     MotionTask Inputs/ControllerTags.arRealAxisAdmin[22].Axis.NcToPlc <-> Outputs/ToPlc
//     MotionTask Outputs/ControllerTags.arRealAxisAdmin[22].Axis.PlcToNc <-> Inputs/FromPlc
//   PLC1/PLC1 Instance <-> NC-Task 1 SAF/Axes/Counter 23
//     MotionTask Inputs/ControllerTags.arRealAxisAdmin[23].Axis.NcToPlc <-> Outputs/ToPlc
//     MotionTask Outputs/ControllerTags.arRealAxisAdmin[23].Axis.PlcToNc <-> Inputs/FromPlc
//   PLC1/PLC1 Instance <-> NC-Task 1 SAF/Axes/Counter 24
//     MotionTask Inputs/ControllerTags.arRealAxisAdmin[24].Axis.NcToPlc <-> Outputs/ToPlc
//     MotionTask Outputs/ControllerTags.arRealAxisAdmin[24].Axis.PlcToNc <-> Inputs/FromPlc
//   PLC1/PLC1 Instance <-> NC-Task 1 SAF/Axes/Counter 25
//     MotionTask Inputs/ControllerTags.arRealAxisAdmin[25].Axis.NcToPlc <-> Outputs/ToPlc
//     MotionTask Outputs/ControllerTags.arRealAxisAdmin[25].Axis.PlcToNc <-> Inputs/FromPlc
//   PLC1/PLC1 Instance <-> NC-Task 1 SAF/Axes/Counter 26
//     MotionTask Inputs/ControllerTags.arRealAxisAdmin[26].Axis.NcToPlc <-> Outputs/ToPlc
//     MotionTask Outputs/ControllerTags.arRealAxisAdmin[26].Axis.PlcToNc <-> Inputs/FromPlc
//   PLC1/PLC1 Instance <-> NC-Task 1 SAF/Axes/Counter 27
//     MotionTask Inputs/ControllerTags.arRealAxisAdmin[27].Axis.NcToPlc <-> Outputs/ToPlc
//     MotionTask Outputs/ControllerTags.arRealAxisAdmin[27].Axis.PlcToNc <-> Inputs/FromPlc
//   PLC1/PLC1 Instance <-> NC-Task 1 SAF/Axes/Counter 28
//     MotionTask Inputs/ControllerTags.arRealAxisAdmin[28].Axis.NcToPlc <-> Outputs/ToPlc
//     MotionTask Outputs/ControllerTags.arRealAxisAdmin[28].Axis.PlcToNc <-> Inputs/FromPlc
//   PLC1/PLC1 Instance <-> NC-Task 1 SAF/Axes/Counter 29
//     MotionTask Inputs/ControllerTags.arRealAxisAdmin[29].Axis.NcToPlc <-> Outputs/ToPlc
//     MotionTask Outputs/ControllerTags.arRealAxisAdmin[29].Axis.PlcToNc <-> Inputs/FromPlc
//   PLC1/PLC1 Instance <-> NC-Task 1 SAF/Axes/Counter 3
//     MotionTask Inputs/ControllerTags.arRealAxisAdmin[3].Axis.NcToPlc <-> Outputs/ToPlc
//     MotionTask Outputs/ControllerTags.arRealAxisAdmin[3].Axis.PlcToNc <-> Inputs/FromPlc
//   PLC1/PLC1 Instance <-> NC-Task 1 SAF/Axes/Counter 30
//     MotionTask Inputs/ControllerTags.arRealAxisAdmin[30].Axis.NcToPlc <-> Outputs/ToPlc
//     MotionTask Outputs/ControllerTags.arRealAxisAdmin[30].Axis.PlcToNc <-> Inputs/FromPlc
//   PLC1/PLC1 Instance <-> NC-Task 1 SAF/Axes/Counter 31
//     MotionTask Inputs/ControllerTags.arRealAxisAdmin[31].Axis.NcToPlc <-> Outputs/ToPlc
//     MotionTask Outputs/ControllerTags.arRealAxisAdmin[31].Axis.PlcToNc <-> Inputs/FromPlc
//   PLC1/PLC1 Instance <-> NC-Task 1 SAF/Axes/Counter 32
//     MotionTask Inputs/ControllerTags.arRealAxisAdmin[32].Axis.NcToPlc <-> Outputs/ToPlc
//     MotionTask Outputs/ControllerTags.arRealAxisAdmin[32].Axis.PlcToNc <-> Inputs/FromPlc
//   PLC1/PLC1 Instance <-> NC-Task 1 SAF/Axes/Counter 33
//     MotionTask Inputs/ControllerTags.arRealAxisAdmin[33].Axis.NcToPlc <-> Outputs/ToPlc
//     MotionTask Outputs/ControllerTags.arRealAxisAdmin[33].Axis.PlcToNc <-> Inputs/FromPlc
//   PLC1/PLC1 Instance <-> NC-Task 1 SAF/Axes/Counter 34
//     MotionTask Inputs/ControllerTags.arRealAxisAdmin[34].Axis.NcToPlc <-> Outputs/ToPlc
//     MotionTask Outputs/ControllerTags.arRealAxisAdmin[34].Axis.PlcToNc <-> Inputs/FromPlc
//   PLC1/PLC1 Instance <-> NC-Task 1 SAF/Axes/Counter 35
//     MotionTask Inputs/ControllerTags.arRealAxisAdmin[35].Axis.NcToPlc <-> Outputs/ToPlc
//     MotionTask Outputs/ControllerTags.arRealAxisAdmin[35].Axis.PlcToNc <-> Inputs/FromPlc
//   PLC1/PLC1 Instance <-> NC-Task 1 SAF/Axes/Counter 36
//     MotionTask Inputs/ControllerTags.arRealAxisAdmin[36].Axis.NcToPlc <-> Outputs/ToPlc
//     MotionTask Outputs/ControllerTags.arRealAxisAdmin[36].Axis.PlcToNc <-> Inputs/FromPlc
//   PLC1/PLC1 Instance <-> NC-Task 1 SAF/Axes/Counter 37
//     MotionTask Inputs/ControllerTags.arRealAxisAdmin[37].Axis.NcToPlc <-> Outputs/ToPlc
//     MotionTask Outputs/ControllerTags.arRealAxisAdmin[37].Axis.PlcToNc <-> Inputs/FromPlc
//   PLC1/PLC1 Instance <-> NC-Task 1 SAF/Axes/Counter 38
//     MotionTask Inputs/ControllerTags.arRealAxisAdmin[38].Axis.NcToPlc <-> Outputs/ToPlc
//     MotionTask Outputs/ControllerTags.arRealAxisAdmin[38].Axis.PlcToNc <-> Inputs/FromPlc
//   PLC1/PLC1 Instance <-> NC-Task 1 SAF/Axes/Counter 39
//     MotionTask Inputs/ControllerTags.arRealAxisAdmin[39].Axis.NcToPlc <-> Outputs/ToPlc
//     MotionTask Outputs/ControllerTags.arRealAxisAdmin[39].Axis.PlcToNc <-> Inputs/FromPlc
//   PLC1/PLC1 Instance <-> NC-Task 1 SAF/Axes/Counter 4
//     MotionTask Inputs/ControllerTags.arRealAxisAdmin[4].Axis.NcToPlc <-> Outputs/ToPlc
//     MotionTask Outputs/ControllerTags.arRealAxisAdmin[4].Axis.PlcToNc <-> Inputs/FromPlc
//   PLC1/PLC1 Instance <-> NC-Task 1 SAF/Axes/Counter 40
//     MotionTask Inputs/ControllerTags.arRealAxisAdmin[40].Axis.NcToPlc <-> Outputs/ToPlc
//     MotionTask Outputs/ControllerTags.arRealAxisAdmin[40].Axis.PlcToNc <-> Inputs/FromPlc
//   PLC1/PLC1 Instance <-> NC-Task 1 SAF/Axes/Counter 5
//     MotionTask Inputs/ControllerTags.arRealAxisAdmin[5].Axis.NcToPlc <-> Outputs/ToPlc
//     MotionTask Outputs/ControllerTags.arRealAxisAdmin[5].Axis.PlcToNc <-> Inputs/FromPlc
//   PLC1/PLC1 Instance <-> NC-Task 1 SAF/Axes/Counter 6
//     MotionTask Inputs/ControllerTags.arRealAxisAdmin[6].Axis.NcToPlc <-> Outputs/ToPlc
//     MotionTask Outputs/ControllerTags.arRealAxisAdmin[6].Axis.PlcToNc <-> Inputs/FromPlc
//   PLC1/PLC1 Instance <-> NC-Task 1 SAF/Axes/Counter 7
//     MotionTask Inputs/ControllerTags.arRealAxisAdmin[7].Axis.NcToPlc <-> Outputs/ToPlc
//     MotionTask Outputs/ControllerTags.arRealAxisAdmin[7].Axis.PlcToNc <-> Inputs/FromPlc
//   PLC1/PLC1 Instance <-> NC-Task 1 SAF/Axes/Counter 8
//     MotionTask Inputs/ControllerTags.arRealAxisAdmin[8].Axis.NcToPlc <-> Outputs/ToPlc
//     MotionTask Outputs/ControllerTags.arRealAxisAdmin[8].Axis.PlcToNc <-> Inputs/FromPlc
//   PLC1/PLC1 Instance <-> NC-Task 1 SAF/Axes/Counter 9
//     MotionTask Inputs/ControllerTags.arRealAxisAdmin[9].Axis.NcToPlc <-> Outputs/ToPlc
//     MotionTask Outputs/ControllerTags.arRealAxisAdmin[9].Axis.PlcToNc <-> Inputs/FromPlc
//   PLC1/PLC1 Instance <-> NC-Task 1 SAF/Axes/Puller
//     MotionTask Inputs/ControllerTags.arRealAxisAdmin[47].Axis.NcToPlc <-> Outputs/ToPlc
//     MotionTask Outputs/ControllerTags.arRealAxisAdmin[47].Axis.PlcToNc <-> Inputs/FromPlc
//   PLC1/PLC1 Instance <-> NC-Task 1 SAF/Axes/V_Master
//     MotionTask Inputs/ControllerTags.arVirtualAxisAdmin[1].Axis.NcToPlc <-> Outputs/ToPlc
//     MotionTask Outputs/ControllerTags.arVirtualAxisAdmin[1].Axis.PlcToNc <-> Inputs/FromPlc
//   PLC1/PLC1 Instance <-> NC-Task 1 SAF/Axes/V_Master2
//     MotionTask Inputs/ControllerTags.arVirtualAxisAdmin[2].Axis.NcToPlc <-> Outputs/ToPlc
//     MotionTask Outputs/ControllerTags.arVirtualAxisAdmin[2].Axis.PlcToNc <-> Inputs/FromPlc
//   PLC1/PLC1 Instance <-> NC-Task 1 SAF/Axes/eAxis1
//     PlcTask1 Inputs/ControllerTags.EncoderAxis[1].NcToPlc <-> Outputs/ToPlc
//     PlcTask1 Outputs/ControllerTags.EncoderAxis[1].PlcToNc <-> Inputs/FromPlc

CONFIGURATION PLC1
    RESOURCE PLC ON TwinCAT3
        TASK CommunicationTask(INTERVAL := T#10ms, PRIORITY := 16);
        TASK IOTask(INTERVAL := T#2ms, PRIORITY := 8);
        TASK MotionTask(INTERVAL := T#2ms, PRIORITY := 6);
        TASK PlcTask1(INTERVAL := T#10ms, PRIORITY := 14);
        PROGRAM EtherCatStates WITH CommunicationTask : EtherCatStates;
        PROGRAM Socket WITH CommunicationTask : Socket;
        PROGRAM IO_Mapping WITH IOTask : IO_Mapping;
        PROGRAM MotionControl WITH MotionTask : MotionControl;
        PROGRAM UN01 WITH PlcTask1 : UN01;
    END_RESOURCE
END_CONFIGURATION

// ---- Data-Types/User-Defined/Condition.TcDUT
TYPE Condition :
(
	Clearing,
	Starting,
	Stopping,
	Aborting,
	Holding,
	UnHolding,
	Suspending,
	UnSuspending,
	Resetting,
    Clearing_Done,
	Starting_Done,
	Stopping_Done,
	Aborting_Done,
	Holding_Done,
	UnHolding_Done,
	Suspending_Done,
	UnSuspending_Done,
	Resetting_Done
) INT;
END_TYPE

// ---- Data-Types/User-Defined/Seq_Status.TcDUT
TYPE Seq_Status :
(
	Seq_Starting:=110,
	Seq_Resetting:=10,
	Seq_Stopping:=900,
	Seq_ClearingDone,
	Seq_StartingDone,
	Seq_StoppingDone:=1000,
	Seq_AbortingDone,
	Seq_SuspendingDone,
	Seq_ResettingDone:=100
)INT;
END_TYPE

// ---- Data-Types/User-Defined/SocketConnect.TcDUT
TYPE SocketConnect :
(
	SocketInit:=0,
	SocketConnect,
	SocketSend,
	SocketRecive,
	SocketClose,
	SocketReset
)INT;
END_TYPE

// ---- Data-Types/User-Defined/UDT_BinBelt.TcDUT
TYPE UDT_BinBelt :
STRUCT
	bin: ARRAY [1..64] OF UDT_Bin;
END_STRUCT
END_TYPE

// ---- Data-Types/User-Defined/UDT_BoxList.TcDUT
TYPE UDT_BoxList :
STRUCT
	Box: ARRAY[0..64] OF UDT_BOX;
END_STRUCT
END_TYPE

// ---- Data-Types/User-Defined/UDT_Hmi_AxisView.TcDUT
TYPE UDT_Hmi_AxisView :
STRUCT
	 Enable: BOOL;
	 JogP: BOOL;
	 JogN: BOOL;
	 MoveReal: BOOL;
	 MoveAbs: BOOL;
	 ActPos: LREAL;
	 Homed: BOOL;
	 Active: BOOL;
END_STRUCT
END_TYPE

// ---- Data-Types/User-Defined/UDT_Hmi_OEE.TcDUT
TYPE UDT_Hmi_OEE :
STRUCT
	OEE: REAL;
	PlannedTime: DINT;
	UsableTime: DINT;
	Usability :REAL;
	DesignSpeed: REAL;
	AverageSpeed: REAL;
	GoodCount: DINT;
	NogoodCount: DINT;
	Performance: REAL;
	Quality: REAL;
	Active: BOOL;
	Reset: BOOL;
	
	ClearingTime: DINT;//清除中
	StoppedTime: DINT;//已停机
	StartingTime: DINT;//启动中
	IdleTime: DINT;//空闲中
	SuspendedTime: DINT;//挂起
	ExecuteTime: DINT;//执行中
	StoppingTime: DINT;//停机中
	AbortingTime: DINT;//终止中
	AbortedTime: DINT;//已终止
	HoldingTime: DINT;//暂停中
	HeldTime: DINT;//已暂停
	UnHoldingTime: DINT;//解除暂停中
	SuspendingTime: DINT;//挂起中
	UnSuspendingTime: DINT;//解除挂起
	ResettingTime: DINT;//重置中
	CompletingTime: DINT;//结束中
	CompleteTime: DINT;//已完成
	
	CounterProcessTime: ARRAY [1..40] OF DINT;
	DropProcessTime: ARRAY [1..40] OF DINT;
END_STRUCT
END_TYPE

// ---- Data-Types/User-Defined/UDT_Recipe.TcDUT
TYPE UDT_Recipe :
STRUCT	
	user: STRING(23);
	amount: DINT;//需要生产的盒数
	counters: ARRAY[1..40] OF UDT_Counters;
END_STRUCT
END_TYPE

// ---- Data-Types/User-Defined/UDT_MS300Output.TcDUT
TYPE UDT_MS300Output :
	STRUCT
		Active: BOOL;
		CmdDone: BOOL;
		Homed: BOOL;
		HomeDone: BOOL;
		ActVel: LREAL;
		ActTorq: LREAL;
		ErrorID: UDINT;
		Error: BOOL;
		PowerOn: BOOL;
		ActPos: LREAL;
		ActModuloPos: LREAL;
		InVelocity: BOOL;
		StopDone: BOOL;
		InGear: BOOL;
		InSync: BOOL; 
		GearOutDone: BOOL;
		CamOutDone: BOOL;
		SetPosDone: BOOL;
		SelectCamTableDone: BOOL; 
		StandStill: BOOL;
		
        ReadyToSwitchOn: BOOL;
		SwitchOn: BOOL;
		OperationEnable: BOOL;
		Fault: BOOL;
		VoltageEnable: BOOL;
		QuickStop: BOOL;
		SwitchOnDisabled: BOOL;
		Warning: BOOL;
		Reserved: BOOL;
		Remote: BOOL;
		TargetReached: BOOL;
		InternalLimitActive: BOOL;
		Operation: BOOL;

		
		
		
	END_STRUCT
END_TYPE

// ---- Data-Types/User-Defined/UDT_MS300Input.TcDUT
TYPE UDT_MS300Input :
STRUCT
  Enable: BOOL;
  Start: BOOL;
  Stop: BOOL;
  Reset: BOOL;
  Vel: INT:=10;
  Acc: LREAL:=100;
  Dec: LREAL:=100;
  Jerk: LREAL;

  RatioNum: LREAL:=1;
  RatioDen: UINT:=1;
	SwitchOn: BOOL;
	EnableVoltage: BOOL;
	QuickStop: BOOL;
	EnableOp: BOOL;
	Operation:BOOL;
	FaultReset: BOOL;
	Halt: BOOL;

  
  
  
  
  
END_STRUCT
END_TYPE

// ---- Data-Types/User-Defined/UDT_DirectMotor.TcDUT
TYPE UDT_DirectMotor :
STRUCT
	Forward: BOOL;
	Backward: BOOL;
END_STRUCT
END_TYPE

// ---- Data-Types/User-Defined/UDT_EL3312.TcDUT
TYPE UDT_EL3312 :
STRUCT
	Status: INT;
	Value: INT;
END_STRUCT
END_TYPE

// ---- Data-Types/User-Defined/UDT_EVENT.TcDUT
TYPE UDT_EVENT :
STRUCT
	ID: ARRAY[1..256] OF BOOL;
END_STRUCT
END_TYPE

// ---- Data-Types/User-Defined/UDT_AxisAdmin.TcDUT
TYPE UDT_AxisAdmin :
STRUCT
	i: UDT_AXISinput;
	o: UDT_AXISOUTPUT;
	Axis: Axis_Ref;
END_STRUCT
END_TYPE

// ---- Data-Types/User-Defined/UDT_AxisInput.TcDUT
TYPE UDT_AxisInput :
STRUCT
  Mode: INT;
  Enable: BOOL;
  MoveAbs: BOOL;
  MoveAdd: BOOL;
  MoveReal: BOOL;
  MoveVel: BOOL;
  Stop: BOOL;
  Home: BOOL;
  Reset: BOOL;
  Pos: LREAL;
  Dist: LREAL;
  Vel: LREAL:=10;
  Acc: LREAL:=100;
  Dec: LREAL:=100;
  Jerk: LREAL;
  StopDec: LREAL:=1000;
  HomeOffset: REAL;
  HomeMode: DINT;
  JogP: BOOL;
  JogN: BOOL;
  JogVel: LREAL:=10;
  JogAcc: LREAL:=100;
  JogDec: LREAL:=100;
  HomeCali: BOOL;
  Direction: MC_Direction;
  GearIn: BOOL;
  GearOut: BOOL;
  CamIn: BOOL;
  CamOut: BOOL;
  RatioNum: LREAL:=1;
  RatioDen: UINT:=1;
  SetPosExe: BOOL;
  SetPosPar: LREAL:=0;
  SelectCamTable: BOOL;
  Disable: BOOL;
  PosRangeTable: ARRAY[1..8] OF ARRAY[1..2] OF LREAL;
END_STRUCT
END_TYPE

// ---- Data-Types/User-Defined/UDT_AxisOutput.TcDUT
TYPE UDT_AxisOutput :
	STRUCT
		Active: BOOL;
		CmdDone: BOOL;
		Homed: BOOL;
		HomeDone: BOOL;
		ActVel: LREAL;
		ActTorq: LREAL;
		ErrorID: UDINT;
		Error: BOOL;
		PowerOn: BOOL;
		ActPos: LREAL;
		ActModuloPos: LREAL;
		InVelocity: BOOL;
		StopDone: BOOL;
		InGear: BOOL;
		InSync: BOOL; 
		InCam: BOOL;
		GearOutDone: BOOL;
		CamOutDone: BOOL;
		SetPosDone: BOOL;
		SelectCamTableDone: BOOL; 
		StandStill: BOOL;
		PosInRange: ARRAY[1..8] OF BOOL;
	END_STRUCT
END_TYPE

// ---- Data-Types/User-Defined/UDT_Box.TcDUT
TYPE UDT_Box :
STRUCT
	PrintData: STRING(23);
	PrintRequest: BOOL;
    amount: DINT;
	Valid :BOOL;
	Drop: BOOL;
	Cut: BOOL;
	Check1: BOOL;
	Check2: BOOL;
	Seal1: BOOL;
	Seal2: BOOL;
	Transfer: BOOL;
	Pick: BOOL;
	Reject: BOOL;
END_STRUCT
END_TYPE

// ---- Data-Types/User-Defined/UDT_CM_Condition.TcDUT
TYPE UDT_CM_Condition :
STRUCT
	Clearing_Done: BOOL;//清除完成
	Starting_Done: BOOL;//启动完成
	Stopping_Done: BOOL;//停机完成
	Aborting_Done: BOOL;//终止完成
	Holding_Done: BOOL;//暂停完成
	UnHolding_Done: BOOL;//解除暂停完成
	Suspending_Done: BOOL;//挂起完成
	UnSuspending_Done: BOOL;//解除挂起完成
	Resetting_Done: BOOL;//重置完成
END_STRUCT
END_TYPE

// ---- Data-Types/User-Defined/UDT_CylinderAdmin.TcDUT
TYPE UDT_CylinderAdmin :
STRUCT
	i: UDT_CylinderInput;
	o: UDT_CylinderOutput;
END_STRUCT
END_TYPE

// ---- Data-Types/User-Defined/UDT_CylinderInput.TcDUT
TYPE UDT_CylinderInput :
STRUCT
	Mode: BOOL; //模式
	Reset: BOOL; //复位
	ActiveIn: BOOL; //原位
	ActiveOut: BOOL; //工作位
	InSensor: BOOL; //原位检测
	OutSensor: BOOL; //工作位检测
	CheckTime: DINT; //检测时间
	HmiIN: BOOL;
	HmiOut: BOOL;
END_STRUCT
END_TYPE

// ---- Data-Types/User-Defined/UDT_CylinderOutput.TcDUT
TYPE UDT_CylinderOutput :
STRUCT
	ValveIn: BOOL;
	ValveOut: BOOL;
	Error: BOOL;
	ErrorID: DINT;
END_STRUCT
END_TYPE

// ---- Data-Types/User-Defined/UDT_EM_Status.TcDUT
TYPE UDT_EM_Status :
STRUCT
	Selected: BOOL;//启用中
	Faulted: BOOL;
	EnableDone: BOOL;
	DisableDone: BOOL;
	StartExecutionDone: BOOL;
	PrepareExecutionDone: BOOL;
	AbortingDone: BOOL;
	StoppingDone: BOOL;
	FaultResetDone: BOOL;
	HomeDone: BOOL;
	PauseDone: BOOL;
	CycleInStandbyDone: BOOL;
	WarningEvent: BOOL;
	GeneralEvent: BOOL;
	StopEvent: BOOL;	
END_STRUCT
END_TYPE

// ---- Data-Types/User-Defined/UDT_EM_Cmd.TcDUT
TYPE UDT_EM_Cmd :
STRUCT
	Mode: DINT;
	Enable: BOOL;
	Disable: BOOL;
	StartExecution: bool;
	PrepareExecution: BOOL;
	Abort: BOOL;
	Stop: BOOL;
	FaultReset: BOOL;
	Home: BOOL;
	Pause: BOOL;
	CycleInStandby: BOOL;
	ResumeFromPause: BOOL;
	ResumeFromCycleInStandby: BOOL;
END_STRUCT
END_TYPE

// ---- Data-Types/User-Defined/UDT_Counters.TcDUT
TYPE UDT_Counters :
STRUCT
	ID: DINT; //当前药品ID
	Quantity: DINT;//当前站需要数的数量
END_STRUCT
END_TYPE

// ---- Data-Types/User-Defined/UDT_Hmi_Input.TcDUT
TYPE UDT_Hmi_Input :
STRUCT
	Reset: BOOL;//触摸屏复位
	Start: BOOL;//触摸屏启动
	Hold: BOOL;//触摸屏暂停	
	Stop: BOOL;//触摸屏停止
	ClearFault: BOOL;//触摸屏错位清除	Belt
	ModifyRecipe: BOOL; //更换配方请求,为1时PLC将输入的配方写入,并在配方输出中变更
END_STRUCT
END_TYPE

// ---- Data-Types/User-Defined/UDT_Hmi_Output.TcDUT
TYPE UDT_Hmi_Output :
STRUCT
	RecipeModifyDone: BOOL;//PLC配方切换完成	
	RecipeProduction: BOOL;//生产中
	RecipeComplete: BOOL;//生产完成	
	RecipeEmplty: BOOL; //
	InQuantity: DINT;//实时反馈当前生产的数量
	OutQuantity: DINT;//实时反馈当前生产的数量
	Counters: ARRAY[1..40]OF UDT_Counters;//当前40个工位粒机信息                                 
END_STRUCT
END_TYPE

// ---- Data-Types/User-Defined/UDT_MS300Admin.TcDUT
TYPE UDT_MS300Admin :
STRUCT
	MS300: UDT_MS300_REF;
    i: UDT_MS300Input;
	o: UDT_MS300OUTPUT;
END_STRUCT
END_TYPE

// ---- Data-Types/User-Defined/UDT_MS300_REF.TcDUT
TYPE UDT_MS300_REF :
STRUCT
	StatusWord AT %I* : UINT;
	VeloDemand AT %I*: INT;
	ModeDisplay AT %I*: SINT;
	ControlWord AT %Q* :UINT;
	TargetVelo AT %Q* :INT;
	ModeOperation AT %Q* :SINT;
END_STRUCT
END_TYPE

// ---- Data-Types/User-Defined/UDT_Bin.TcDUT
TYPE UDT_Bin :
STRUCT
	lrlatchPos: LREAL;
	bValid: BOOL;
	bReject: BOOL;
	arDrop: ARRAY[1..64] OF BOOL;
	Name: STRING(23);
	Amount: DINT;
END_STRUCT
END_TYPE

// ---- Data-Types/User-Defined/UDT_BinList.TcDUT
TYPE UDT_BinList :
STRUCT
	Bin: ARRAY[0..255] OF  UDT_Bin;
	arWorkPos: ARRAY[1..40] OF LREAL;
	arInRang: ARRAY[1..40] OF BOOL;
	Reset: BOOL;
END_STRUCT
END_TYPE

// ---- Data-Types/User-Defined/UDT_Scara.TcDUT
TYPE UDT_Scara :
STRUCT
	i: UDT_Scara_DI;
	o: UDT_Scara_DO;
	Busy: BOOL;
	DI_: ARRAY[1..8] OF ARRAY[1..8] OF BOOL;
	DO_: ARRAY[1..8] OF ARRAY[1..8] OF BOOL;
END_STRUCT
END_TYPE

// ---- Data-Types/User-Defined/UDT_Scara_DI.TcDUT
TYPE UDT_Scara_DI :
STRUCT
	Shutdown: BOOL;
	Estop: BOOL;
	Auto: BOOL;
	T2: BOOL;
	Start: BOOL;
	Hold: BOOL;
	Unhold: BOOL;
	Ready: BOOL;
	Stop: BOOL;
	Reset: BOOL;
	ProFaultClear: BOOL;
	ProPick: BOOL;
	ProDepart: BOOL;
	ProPut: BOOL;
	FuctionReset: BOOL;
	LoopRun: BOOL;
	LoopStop: BOOL;
END_STRUCT
END_TYPE

// ---- Data-Types/User-Defined/UDT_Scara_DO.TcDUT
TYPE UDT_Scara_DO :
STRUCT
    Error: BOOL;
	Enable: BOOL;
	ProRunning: BOOL;
	ProFault: BOOL;
	ProPickDone: BOOL;
	ProPutDone: BOOL;
	ProDepartDone: BOOL;
	Held: BOOL;
	InPos: BOOL;
	ProStopped: BOOL;
	FuctionHold: BOOL;
    loopRunActive :BOOL;
	LoopStopDone: BOOL;
	ResettingDone: BOOL;
END_STRUCT
END_TYPE

// ---- Data-Types/User-Defined/UDT_SensorAdmin.TcDUT
TYPE UDT_SensorAdmin :
STRUCT
	i: UDT_SENSORINPUT;
	o: UDT_SENSOROUTPUT;
END_STRUCT
END_TYPE

// ---- Data-Types/User-Defined/UDT_SensorInput.TcDUT
TYPE UDT_SensorInput :
STRUCT
	Link: BOOL;
	FilterTime: DINT;
END_STRUCT
END_TYPE

// ---- Data-Types/User-Defined/UDT_SensorOutput.TcDUT
TYPE UDT_SensorOutput :
STRUCT
	Value: BOOL;
END_STRUCT
END_TYPE

// ---- Data-Types/User-Defined/UDT_UnitAdmin.TcDUT
TYPE UDT_UnitAdmin :
STRUCT
	Cmd: UDT_Unit_Cmd;
	Sts: UDT_Unit_Status;
	EM_Selected: ARRAY[0..64]OF BOOL;
	EM_Clearing_Done: ARRAY[0..64]OF BOOL;//清除中
	EM_Starting_Done: ARRAY[0..64]OF BOOL;//启动中
	EM_Stopping_Done: ARRAY[0..64]OF BOOL;//停机中
	EM_Aborting_Done: ARRAY[0..64]OF BOOL;//终止中
	EM_Holding_Done: ARRAY[0..64]OF BOOL;//暂停中
	EM_UnHolding_Done: ARRAY[0..64]OF BOOL;//解除暂停中
	EM_Suspending_Done: ARRAY[0..64]OF BOOL;//挂起中
	EM_UnSuspending_Done: ARRAY[0..64]OF BOOL;//解除挂起
	EM_Resetting_Done: ARRAY[0..64]OF BOOL;//重置中
	EM_Fault: ARRAY[0..64] OF BOOL;
	EM_Warning: ARRAY[0..64] OF BOOL;
	GeneralEvent: ARRAY[0..64] OF DINT;
	WarningEvent: ARRAY[0..64] OF DINT;
	StopEvent: ARRAY[0..64] OF DINT;  	
END_STRUCT
END_TYPE

// ---- Data-Types/User-Defined/UDT_Unit_Cmd.TcDUT
TYPE UDT_Unit_Cmd :
STRUCT
	Mode: DINT;//模式 0手动,1自动
	Reset: BOOL;//复位
	Start: BOOL;//启动
	Stop: BOOL;//停止
	Hold: BOOL;//暂停
	UnHold: BOOL;//解除暂停
	Suspend: BOOL;//挂起
	UnSuspend: BOOL;//解除挂起
	Abort: BOOL;//中止
	Clear: BOOL;//清除故障
END_STRUCT
END_TYPE

// ---- Data-Types/User-Defined/UDT_Unit_Status.TcDUT
TYPE UDT_Unit_Status :
STRUCT
	Clearing: BOOL;//清除中
	Stopped: BOOL;//已停机
	Starting: BOOL;//启动中
	Idle: BOOL;//空闲中
	Suspended: BOOL;//挂起
	Execute: BOOL;//执行中
	Stopping: BOOL;//停机中
	Aborting: BOOL;//终止中
	Aborted: BOOL;//已终止
	Holding: BOOL;//暂停中
	Held: BOOL;//已暂停
	UnHolding: BOOL;//解除暂停中
	Suspending: BOOL;//挂起中
	UnSuspending: BOOL;//解除挂起
	Resetting: BOOL;//重置中
	Completing: BOOL;//结束中
	Complete: BOOL;//已完成
END_STRUCT
END_TYPE

// ---- Data-Types/User-Defined/UDT_VacuumAdmin.TcDUT
TYPE UDT_VacuumAdmin :
STRUCT
	i: UDT_VacuumInput;
	o: UDT_VacuumOutput;
END_STRUCT
END_TYPE

// ---- Data-Types/User-Defined/UDT_VacuumInput.TcDUT
TYPE UDT_VacuumInput :
STRUCT
	ActiveIN: BOOL; 
	ActiveOut: BOOL;
	Sensor: BOOL;
	CheckTime: DINT;
	BlowTime: DINT;
	HmiIN: BOOL;
	HmiOut: BOOL;
	Reset: BOOL;
END_STRUCT
END_TYPE

// ---- Data-Types/User-Defined/UDT_VacuumOutput.TcDUT
TYPE UDT_VacuumOutput :
STRUCT
	ValveIn: BOOL;
	ValveOut: BOOL;
	Error: BOOL;
	ErrorID: DINT;
END_STRUCT
END_TYPE

// ---- POUs/GVLs/ControllerTags.TcGVL
VAR_GLOBAL
	UN01_MachineStateModel: PackMlv3_StateModel;
	Unit01: UDT_UnitAdmin;	
	
	UN02_MachineStateModel: PackMlv3_StateModel;
	Unit02: UDT_UnitAdmin;	
	HMI_AlarmMute: BOOL;//报警消音
	HMI_Input:  UDT_Hmi_Input; //远程触摸屏发送数据给设备	
	HMI_Output:  UDT_Hmi_Output; //当前生产的配方反馈给触摸屏
	HMI_Recipe: UDT_Recipe;
	RecipeBuffer: UDT_Recipe;

	arRealAxisAdmin: ARRAY[1..65] OF UDT_AXISADMIN;//实际轴
	arVirtualAxisAdmin: ARRAY[1..65] OF UDT_AXISADMIN;//虚拟轴
	arMS300Admin: ARRAY[1..1] OF UDT_MS300Admin;
	arDropCylinder: ARRAY[1..40] OF UDT_CylinderAdmin;//料仓落料气缸
	arHighSensor: ARRAY[1..40] OF UDT_SensorAdmin;//料仓高料位传感器
	arLowSensor: ARRAY[1..40] OF UDT_SensorAdmin;//料仓低料位传感器
	arDropSensor: ARRAY[1..40] OF UDT_SensorAdmin;//料仓低料位传感器
	arCounters: ARRAY[1..40] OF AOI_CountersAdmin;//料仓控制
    HMI_StopEvent: ARRAY[0..40] OF UDT_EVENT;
	HMI_GeneralEvent: ARRAY[0..10] OF UDT_EVENT;//常规信息
	HMI_WarningEvent: ARRAY[0..10] OF UDT_EVENT;//非停机报警信息
	
	arDropBufferCyclinder: ARRAY[0..10] OF UDT_CylinderAdmin;

	arPackCylinder: ARRAY[1..60] OF UDT_CylinderAdmin;//包装系统气缸组
	arPackVacuum: ARRAY[1..60] OF UDT_VacuumAdmin;//包装系统真空组
	arPackSensor: ARRAY[1..60] OF UDT_SensorAdmin;//包装系统真空组
	arPackMotor: ARRAY[1..16] OF UDT_directMotor;//调速马达
	arPackHeatRealy: ARRAY[1..16] OF BOOL;//加热固态继电器
	EncoderAxis: ARRAY[1..16] OF Axis_Ref;//编码器轴
	(*digital input *)
	EL1008 AT%I* : ARRAY[1..64,1..8] OF BOOL;
	(*digital output*)
	EL2008 AT%Q* : ARRAY[1..64,1..8] OF BOOL;	
	CPX8_1 AT%I* : ARRAY[1..64,1..8] OF BOOL;
	CPX8_2 AT%I* : ARRAY[1..64,1..8] OF BOOL;	
	WPI_1 AT%Q* : ARRAY[1..64,1..8] OF BOOL;
	WPI_2 AT%Q* : ARRAY[1..64,1..8] OF BOOL;
	WPI_3 AT%Q* : ARRAY[1..64,1..8] OF BOOL;
	EL3312 AT%I* : ARRAY[1..16,1..2] OF UDT_EL3312;
	
	DI_: ARRAY [1..64,1..8] OF  AOI_DI;
	DO_: ARRAY [1..64,1..8] OF  AOI_DO;
	
	glb_BinBelt1: UDT_BinBelt;
	glb_BinBelt2: UDT_BinBelt;	
	glb_BinBelt3: UDT_BinBelt;	
	glb_BinBelt4_5: UDT_BinBelt;
	glb_RecipeTotalBin: INT;

	
	glb_AllCountersInitDone: BOOL;
	glb_Un01Box: UDT_BOXLIST;
	glb_rMainBeltSpeed: REAL;//主线速度
	glb_bModeSwitch_UN01: BOOL;//模式选择
	glb_bStartButton_UN01: BOOL;//启动按钮
	glb_bStopButton_UN01: BOOL;//停止按钮
	glb_diEstopButton_UN01: DINT;//急停按钮
	glb_bResetButton_UN01: BOOL;//复位按钮
	glb_bAirFeedback_UN01: ARRAY[1..8] OF BOOL;//气压反馈
	glb_bStartBottonLight_UN01: BOOL;//启动按钮指示灯
	glb_bStopBottonLight_UN01: BOOL;//停止按钮指示灯
	glb_bResetBottonLight_UN01: BOOL;//复位按钮指示灯
	
	glb_arLightRelay_UN01: ARRAY[1..16] OF BOOL;//数粒系统设备照明继电器
    glb_arLightRed_UN01: ARRAY[1..8] OF BOOL;//三色灯红灯
    glb_arLightYellow_UN01: ARRAY[1..8] OF BOOL;//三色灯黄灯
    glb_arLightGreen_UN01: ARRAY[1..8] OF BOOL;//三色灯绿灯
    glb_arLightAlarm_UN01: ARRAY[1..8] OF BOOL;//三色灯蜂鸣器		
	glb_arSafeRelayNo_UN01: ARRAY[1..8] OF BOOL;;//安全继电器反馈	
	
	glb_bPackAirValve_UN01: BOOL;//总装罐气阀开关
	glb_bCounterAirValve_UN01: BOOL;//数粒气阀开关
	glb_diBeltObjCnt: DINT; //数粒系统中半成品数量
	glb_bUnit01BoxEmpty: BOOL;//前端纸盒全空
	glb_bUnit01BoxNotReady: BOOL;//前端纸盒未就绪
	
	glb_lrMasterTargetCnt: LREAL;//计算主轴的数量
	glb_lrBelt1TargetCnt: LREAL;//计算配方生产完成后belt1的数量	
	glb_lrBelt2TargetCnt: LREAL;//计算配方生产完成后belt2的数量	
	glb_lrBelt3TargetCnt: LREAL;//计算配方生产完成后belt3的数量	
	glb_lrBoxTargetCnt: LREAL;//计算配方生产完成拉盒数量

	glb_lrMasterWrkCnt: LREAL;//计算主轴的数量
	glb_lrBelt1WrkCnt: LREAL;//计算配方生产完成后belt1的数量	
	glb_lrBelt2WrkCnt: LREAL;//计算配方生产完成后belt2的数量	
	glb_lrBelt3WrkCnt: LREAL;//计算配方生产完成后belt3的数量	
	glb_lrBoxWrkCnt: LREAL;//计算配方生产完成拉盒数量

    glb_lrBelt3ValidCnt: LREAL;//belt3的产品数量
	
	glb_bSafetyReset: BOOL;//安全继电器复位
	arSafeDoorSts: ARRAY [1..40] OF  BOOL;
//	arEstopSts: ARRAY [1..40] OF  BOOL;

	glb_Un02Box: UDT_BOXLIST;
	glb_CompleteBox: UDT_BOXLIST;
	glb_bModeSwitch_UN02: BOOL;//模式选择
	glb_bStartButton_UN02: BOOL;//启动按钮
	glb_bStopButton_UN02: BOOL;//停止按钮
	glb_diEstopButton_UN02: DINT;//急停按钮
	glb_bResetButton_UN02: BOOL;//复位按钮
	glb_bAirFeedback_UN02: BOOL;
	
	glb_bStartBottonLight_UN02: BOOL;
	glb_bStopBottonLight_UN02: BOOL;
	glb_bResetBottonLight_UN02: BOOL;

    glb_arLightRed_UN02: ARRAY[1..8] OF BOOL;
    glb_arLightYellow_UN02: ARRAY[1..8] OF BOOL;	
    glb_arLightGreen_UN02: ARRAY[1..8] OF BOOL;	
    glb_arLightAlarm_UN02: ARRAY[1..8] OF BOOL;	
		
	ScaraRobot: UDT_Scara;//机器人(*IP 192.168.1.20*)			
	arErrorCodeDrive AT %I*: ARRAY[1..64] OF UINT;
	
	glb_diNogoodFlag_UN01: DINT;//不良标志	
	glb_diGoodFlag_UN01: DINT;//良品标志
	glb_diPullFlag_UN01: DINT;//拉盒信号
	glb_diDropFlag_UN01: DINT;//落药信号
	glb_diCutFlag_Un01: DINT;//冲裁信号	
	glb_diSealFlag_Un01: DINT;//封盒信号
	glb_diTransferFlag_UN01: DINT;//移载抓取信号
    glb_bTransferPutWait_UN01: BOOL;//等待放置
	glb_bUnit02BoxEmpty: BOOL;//后段铝盒全空
	glb_bWaitRobotPick: BOOL;
	glb_bAllSafetyOk: BOOL;
    glb_bTransferPut_UN02: BOOL;//移载放置信号
	glb_diTransferPick_UN02: DINT;//移载抓取信号
	glb_diPrint_UN02: DINT;//喷印标志位	
	glb_BoxTransferBuffer: UDT_BOX;//移载缓冲区信息
	//ethercat状态
	HMI_EtherCat_States1: ARRAY [0..255] OF STRING;
	HMI_EtherCat_States2: ARRAY [0..255] OF STRING;
	HMI_EtherCat_Name1: ARRAY [0..255] OF STRING;
	HMI_EtherCat_Name2: ARRAY [0..255] OF STRING;
	glb_bDevice1AllOP: BOOL;
	glb_bDevice2AllOP: BOOL;
		
	glb_AllAxisHomed_UN01: BOOL;
	glb_AllAxisHomed_UN02: BOOL;	
	glb_BinList: UDT_BInlist;
	glb_DropFlag: ARRAY[1..40] OF BOOL;
	
	glb_TransferCnt: DINT;
	
	
	HMI_LocModeEnable: BOOL;//启用本地配方模式 
    HMI_LocModeInput: UDT_Hmi_Input;//本地配方模式
	HMI_LocModeInput_UN02: UDT_Hmi_Input;//UN02配方模式	
    HMI_HeatTempAct: ARRAY[1..16] OF REAL;
	HMI_SkipTransferPut: BOOL;
	HMI_RecipeReset: BOOL;
	HMI_RecipeAbort: BOOL;
	HMI_RecipeRedo: BOOL;
	// 取消配方
	HMI_RecipCancel: BOOL;
	
	HMI_ClearCounter: ARRAY[1..40] OF BOOL;
	
	HMI_AxisView: ARRAY[1..64] OF UDT_Hmi_AxisView;
	HMI_OEEView: UDT_Hmi_OEE;
	HMI_BoxViewUN01: ARRAY[0..64] OF STRING;
	HMI_BoxViewUN02: ARRAY[0..64] OF STRING;
	HMI_ManualInhibit: ARRAY[0..255] OF BOOL;
	HMI_HeatDisable: BOOL;
	
	HMI_CompleteBox : UDT_BOX;
	HMI_CompleteUpdate: BOOL;
	HMI_Unit02Simulation :BOOL;
	
	HMI_PrinterTest: BOOL; //喷码机测试
	HMI_PrinterConnected: BOOL; //喷码机通讯正常
	HMI_PrinterFault: BOOL; //喷码机喷码失败
	HMI_PrinterTestData: STRING(22):='T/S MADE POSSIBLE';//喷码机反馈字符	
	HMI_PrinterReceiveData: STRING;//喷码机反馈字符
		
	HMI_AutoCut: BOOL;
	HMI_CutCnt: DINT;

	HMI_CountersCntUp: ARRAY[1..40] OF DINT;
	HMI_DisableCntAlarmAll: BOOL;
	HMI_EnbaleCntAlarmAll : BOOL;
	HMI_DisableCntAlarmAll2: BOOL;
	HMI_EnbaleCntAlarmAll2 : BOOL;	
	// 拉膜报警
	glb_MembraneAlarm: BOOL;
END_VAR


VAR_GLOBAL RETAIN
	HMI_SkipCntAlarm: ARRAY[1..40] OF BOOL;
	HMI_CntCheckTime: DINT:=1500;
	HMI_CntCheck: ARRAY[1..40] OF BOOL;
	
	HMI_HomeOffsetBelt: ARRAY[1..16] OF REAL;//皮带原点
	HMI_BeltVelo: ARRAY[1..16] OF REAL:=[16(50)];//皮带速度
	HMI_BeltAcc: ARRAY[1..16] OF REAL:=[16(100)];;//皮带速度
	HMI_BeltDec: ARRAY[1..16] OF REAL:=[16(100)];;//皮带速度
	HMI_CountersVelo: LREAL;
	HMI_CountersAcc: LREAL;
	HMI_CountersDec: LREAL;
	HMI_MasterVelo: LREAL;//主轴速度
	HMI_HeatTempSet: ARRAY[1..16] OF REAL;//加热温度设置
	HMI_SealTime: DINT;//封口时间
	HMI_SealTime2: DINT;//封口时间	
	HMI_arSealTime: array[1..8] of DINT;
	HMI_PullerPara: ARRAY[1..8] OF LREAL;//[1]拉膜长度 [2]拉膜速度
	HMI_PusherPos: ARRAY[1..8] OF LREAL;
	HMI_EMSelectUN01: ARRAY[0..64] OF BOOL;
	HMI_EMSelectUN02: ARRAY[0..64] OF BOOL;
	
	HMI_PrintNo: INT:=11;//打印站位号
	HMI_PrintMaxTime: DINT:=30;//最大打印监控时间
    HMI_PickNo: INT:=7;//抓取站位号	
	
	HMI_DropNo: INT:=2;//落料站位号
	HMI_CutNo: INT:=7;//裁切站位号
	HMI_Check1No: INT:=4;//铝杯检测1站位号
	HMI_Check2No: INT:=5;//铝杯检测2站位号	
	HMI_Seal1No: INT:=10;//封口1站位号
	HMI_Seal2No: INT:=11;//封口2站位号
	HMI_TransferNo: INT:=13;//封口1站位号	
	
	HMI_DropPosOffset: REAL:=-120;
	HMI_B3DropBinNo1: INT:=1;
	HMI_B3DropBinNo2: INT:=14;
	HMI_B3DropBinNo3: INT:=28;
	HMI_B2DropBinNo: INT:=12;
	HMI_B1DropBinNo: INT:=12;	
	
END_VAR

// ---- POUs/EtherCat/EtherCatStates.TcPOU
PROGRAM EtherCatStates
VAR
	Device1_netID AT %I*:Tc2_System.T_AmsNetIdArr;							//硬件网络的AMSnetID
	Device1_nEcMasterDeviceId AT %I*:UINT;		//主站的deviceID
	
    Device1_slaveAddresses    : ARRAY[0..255] OF UINT;						//读取的从站地址（以数组保存）
	Device1_devStates           : ARRAY[0..255] OF ST_EcSlaveState;		//读取的从站状态机
	Device1_slavenames			: ARRAY[0..255] OF T_MaxString;			//读取从站名字
	Device1_nSlaves           : UINT := 0;														//从站个数
    i:INT;
	
	Device1_fb_getalladdr:Tc2_EtherCAT.FB_EcGetAllSlaveAddr;		//读取从站地址的功能块 https://infosys.beckhoff.com/content/1033/tcplclib_tc2_ethercat/9007199311752331.html?id=8671424095593379685
	Device1_fb_getallstate:Tc2_EtherCAT.FB_EcGetAllSlaveStates;		//读取从站状态机的功能块 https://infosys.beckhoff.com/content/1033/tcplclib_tc2_ethercat/9007199311770635.html?id=2217456128990928132
	Device1_fb_getallname: IOF_GetBoxNameByAddr;							//读取从站名称 https://
	ton1: Ton;
	bExecute: BOOL;
	
	
	Device2_netID AT %I*:Tc2_System.T_AmsNetIdArr;							//硬件网络的AMSnetID
	Device2_nEcMasterDeviceId AT %I*:UINT;		//主站的deviceID
	
    Device2_slaveAddresses    : ARRAY[0..255] OF UINT;						//读取的从站地址（以数组保存）
	Device2_devStates           : ARRAY[0..255] OF ST_EcSlaveState;		//读取的从站状态机
	Device2_slavenames			: ARRAY[0..255] OF T_MaxString;			//读取从站名字
	Device2_nSlaves           : UINT := 0;														//从站个数
    k:INT;
	
	Device2_fb_getalladdr:Tc2_EtherCAT.FB_EcGetAllSlaveAddr;		//读取从站地址的功能块 https://infosys.beckhoff.com/content/1033/tcplclib_tc2_ethercat/9007199311752331.html?id=8671424095593379685
	Device2_fb_getallstate:Tc2_EtherCAT.FB_EcGetAllSlaveStates;		//读取从站状态机的功能块 https://infosys.beckhoff.com/content/1033/tcplclib_tc2_ethercat/9007199311770635.html?id=2217456128990928132
	Device2_fb_getallname: IOF_GetBoxNameByAddr;							//读取从站名称 https://
	
	
	
	
	iDevice2OPCnt: INT;
	j: INT;
	iDevice1OPCnt: INT;
	
	
	fbPlc_Shutdown:	NT_Shutdown;
	bPlcShutDown: BOOL;
END_VAR

ton1(IN:= NOT ton1.Q, PT:= T#2S, Q=> bExecute, ET=> );

Device1_fb_getalladdr(//读取从站地址
	sNetId:= F_CreateAmsNetId(Device1_netID), //网络netID
	pAddrBuf:= ADR(Device1_slaveAddresses), //寄存器地址
	cbBufLen:= SIZEOF(Device1_slaveAddresses), 
	bExecute:= bExecute, 
	nSlaves=> Device1_nSlaves);//从站个数
	
Device1_fb_getallstate(//读取从站状态机
	sNetId:= F_CreateAmsNetId(Device1_netID), //网络地址
	pStateBuf:= ADR(Device1_devStates), //寄存器地址
	cbBufLen:= SIZEOF(Device1_devStates), 
	bExecute:= bExecute, 
	nSlaves=> );

Device1_fb_getallname(//读取从站名称
	NETID:= , 
	DEVICEID:=Device1_nEcMasterDeviceId, //device number
	BOXADDR:=  Device1_slaveAddresses[j], //从站号
	BOXNAME=> Device1_slavenames[j]);//返回从站名

IF Device1_slaveAddresses[j]>0 AND NOT Device1_fb_getallname .start THEN//反复触发功能块
	Device1_fb_getallname.START:=TRUE;
ELSIF Device1_slaveAddresses[j+1]>0 AND NOT Device1_fb_getallname.BUSY THEN
		j:=j+1;
		Device1_fb_getallname.START:=FALSE;
END_IF



Device2_fb_getalladdr(//读取从站地址
	sNetId:= F_CreateAmsNetId(Device2_netID), //网络netID
	pAddrBuf:= ADR(Device2_slaveAddresses), //寄存器地址
	cbBufLen:= SIZEOF(Device2_slaveAddresses), 
	bExecute:= bExecute, 
	nSlaves=> Device2_nSlaves);//从站个数
	
Device2_fb_getallstate(//读取从站状态机
	sNetId:= F_CreateAmsNetId(Device2_netID), //网络地址
	pStateBuf:= ADR(Device2_devStates), //寄存器地址
	cbBufLen:= SIZEOF(Device2_devStates), 
	bExecute:= bExecute, 
	nSlaves=> );

Device2_fb_getallname(//读取从站名称
	NETID:= , 
	DEVICEID:=Device2_nEcMasterDeviceId, //device number
	BOXADDR:=  Device2_slaveAddresses[k], //从站号
	BOXNAME=> Device2_slavenames[k]);//返回从站名

IF Device2_slaveAddresses[k]>0 AND NOT Device2_fb_getallname .start THEN//反复触发功能块
	Device2_fb_getallname.START:=TRUE;
ELSIF Device2_slaveAddresses[k+1]>0 AND NOT Device2_fb_getallname.BUSY THEN
		k:=k+1;
		Device2_fb_getallname.START:=FALSE;
END_IF

iDevice1OPCnt:=0;
FOR i:=0 TO 106 DO
	IF Device2_devStates[i].deviceState=8 THEN
		iDevice1OPCnt:=iDevice1OPCnt+1;
	END_IF
END_FOR
IF iDevice1OPCnt=107 THEN
   glb_bDevice1AllOP:=TRUE;
   ELSE	   
   glb_bDevice1AllOP:=FALSE;
END_IF
iDevice2OPCnt:=0;
FOR i:=0 TO 43 DO
	IF Device1_devStates[i].deviceState=8 THEN
		iDevice2OPCnt:=iDevice2OPCnt+1;
	END_IF
END_FOR

IF iDevice2OPCnt=44 THEN
	glb_bDevice2AllOP:=TRUE;
	ELSE		
	glb_bDevice2AllOP:=FALSE;
END_IF

FOR i:=0 TO 255 DO
   IF BYTE_TO_SINT(Device1_devStates[i].deviceState)=1 THEN
	   HMI_EtherCat_States1[i]:='Init';
   END_IF
   IF BYTE_TO_SINT(Device1_devStates[i].deviceState)=2 THEN
	   HMI_EtherCat_States1[i]:='Pre-OP';
   END_IF
   IF BYTE_TO_SINT(Device1_devStates[i].deviceState)=3 THEN
	   HMI_EtherCat_States1[i]:='Bootstrap';
   END_IF
   IF BYTE_TO_SINT(Device1_devStates[i].deviceState)=4 THEN
	   HMI_EtherCat_States1[i]:='Safe-OP';
   END_IF
   IF BYTE_TO_SINT(Device1_devStates[i].deviceState)=8 THEN
	   HMI_EtherCat_States1[i]:='OK';
   END_IF

   IF BYTE_TO_SINT(Device2_devStates[i].deviceState)=1 THEN
	   HMI_EtherCat_States2[i]:='Init';
   END_IF
   IF BYTE_TO_SINT(Device2_devStates[i].deviceState)=2 THEN
	   HMI_EtherCat_States2[i]:='Pre-OP';
   END_IF
   IF BYTE_TO_SINT(Device2_devStates[i].deviceState)=3 THEN
	   HMI_EtherCat_States2[i]:='Bootstrap';
   END_IF
   IF BYTE_TO_SINT(Device2_devStates[i].deviceState)=4 THEN
	   HMI_EtherCat_States2[i]:='Safe-OP';
   END_IF
   IF BYTE_TO_SINT(Device2_devStates[i].deviceState)=8 THEN
	   HMI_EtherCat_States2[i]:='OK';
   END_IF
   
   HMI_EtherCat_Name1[i]:= Device1_slavenames[i];
   HMI_EtherCat_Name2[i]:= Device2_slavenames[i];
END_FOR



fbPlc_Shutdown(
	NETID:='5.74.170.4.1.1' , 
	DELAY:= , 
	START:= bPlcShutDown, 
	TMOUT:= , 
	BUSY=> , 
	ERR=> , 
	ERRID=> );

END_PROGRAM

// ---- POUs/Socket/Socket.TcPOU
PROGRAM Socket
VAR
	arSocketListen: ARRAY[1..8] OF FB_SocketListen;
	arSocketAccept: ARRAY[1..8] OF FB_SocketAccept;	
	
	arSocketConnect: ARRAY[1..8] OF FB_SocketConnect;
	arSocketReceive: ARRAY[1..8] OF FB_SocketReceive;
    arSocketSend: ARRAY[1..8] OF FB_SocketSend;	
	arSocketClose: ARRAY[1..8] OF FB_SocketClose;	
		
	arListen: ARRAY[1..8] OF BOOL;
	arhlistener: ARRAY[1..8] OF  T_HSOCKET;

	wReceiveDataBuffer: ARRAY[0..127] OF WORD;
	wSendDataBuffer: ARRAY[0..127] OF WORD;	
	
	wReceiveData: ARRAY[0..127] OF WORD;
	wSendData: ARRAY[0..127] OF WORD;
	wNullData: ARRAY[0..127] OF WORD;
	
	pbyReceiveData: ARRAY [0..255] OF BYTE;;
	pbySendData: ARRAY [0..255] OF BYTE;;
 
	byReceiveData: ARRAY [0..255] OF BYTE;;
	bySendData: ARRAY [0..255] OF BYTE;	
	
	byPrint:  ARRAY [0..MAX_STRING_LENGTH] OF BYTE;
	byPrintAuto:  ARRAY [0..MAX_STRING_LENGTH] OF BYTE;
	byPrintUser:  ARRAY [0..MAX_STRING_LENGTH] OF BYTE;
	
	iSocket: ARRAY[1..8] OF INT;
	arConnectExecute: ARRAY[1..8] OF BOOL;
	arConnectError: ARRAY[1..8] OF BOOL;
	arConnectErrId: ARRAY[1..8] OF UDINT;
	arConnectBusy: ARRAY[1..8] OF BOOL;
		
	arReceiveExecute: ARRAY[1..8] OF BOOL;
	arReceiveError: ARRAY[1..8] OF BOOL;
	arReceiveErrId: ARRAY[1..8] OF UDINT;
	arReceiveBusy: ARRAY[1..8] OF BOOL;
		
	arCloseExecute: ARRAY[1..8] OF BOOL;
	arCloseError: ARRAY[1..8] OF BOOL;
	arCloseErrId: ARRAY[1..8] OF UDINT;
	arCloseBusy: ARRAY[1..8] OF BOOL;
	arhSocket: ARRAY[1..8] OF T_HSOCKET;
	
	arSendExecute: ARRAY[1..8] OF BOOL;

	
	arSendError: ARRAY[1..8] OF BOOL;
	arSendErrId: ARRAY[1..8] OF UDINT;
	arSendBusy: ARRAY[1..8] OF BOOL;
	arTon: ARRAY [1..8] OF Ton;
	arBlink: ARRAY[1..8] OF BLINK;
	
	testString: STRING:='1';
	byteString: BYTE;
	pS: POINTER TO STRING;

	arAccept: ARRAY[1..8] OF bool;
	arListenBusy: ARRAY[1..8] OF bool;
	arAcceptBusy: ARRAY[1..8] OF bool;
	arListenError: ARRAY[1..8] OF bool;
	arAcceptError: ARRAY[1..8] OF bool;

	
	
	byPrintSend: ARRAY [0..MAX_STRING_LENGTH] OF BYTE;
	byPrintReceive: ARRAY [0..MAX_STRING_LENGTH] OF BYTE;


	iPPReceive: INT;
	diReceiveData: DINT;
	iPPSend: INT;
	iPPAccept: INT;

	
	tonFS: TON;
	
	pReceiveString: POINTER TO STRING;
	wSendCnt: WORD;
	
	
	sTestSting: STRING(255);
	arrtestBytearr: ARRAY [0..MAX_STRING_LENGTH] OF BYTE;
	arrToBytearr: ARRAY [0..MAX_STRING_LENGTH] OF BYTE;
	sToBytearrString: T_MaxString;
	sAutoPrintData: STRING(22);
	sTestPrintData: STRING(22);
	bDebugFlag: DINT;
	sTestData: STRING;
	iLen: UINT;
	rViewPrintPos: REAL;
	rPrintPosBuffer: REAL;
END_VAR

//TCP1_Client();
TCP2_Server();
pReceiveString:=ADR(pbyReceiveData);
HMI_PrinterReceiveData:=pReceiveString^;
sTestSting:=BYTEARR_TO_MAXSTRING(in:= arrtestBytearr);
arrToBytearr:=MAXSTRING_TO_BYTEARR(in:= sToBytearrString);

ACTION TCP1_Client:
(*
arSocketConnect[1](
	sSrvNetId:= , 
	sRemoteHost:= '192.168.1.199', 
	nRemotePort:= 3000, 
	bExecute:= arConnectExecute[1] , 
	tTimeout:= T#10S, 
	bBusy=> arConnectBusy[1], 
	bError=> arConnectError[1], 
	nErrId=> arConnectErrId[1], 
	hSocket=> arhSocket[1]);
		
arBlink[1](TimeH:= 1000, TimeL:= 2000, OUT=> );
	
arSocketReceive[1](
	sSrvNetId:= , 
	hSocket:=  arhSocket[1], 
	cbLen:= 255, 
	pDest:= ADR(ReceiveData[1]), 
	bExecute:= arReceiveExecute[1], 
	tTimeout:= T#1S, 
	bBusy=> arReceiveBusy[1], 
	bError=> arReceiveError[1], 
	nErrId=> arReceiveErrId[1], 
	nRecBytes=> );

arSocketSend[1](
	sSrvNetId:= , 
	hSocket:= arhSocket[1], 
	cbLen:=  255, 
	pSrc:= ADR(SendData[1]), 
	bExecute:= arSendExecute[1], 
	tTimeout:= T#1S, 
	bBusy=> arSendBusy[1], 
	bError=> arSendError[1], 
	nErrId=> arSendErrId[1]);	
	
	
arSocketClose[1](
	sSrvNetId:= , 
	hSocket:=  arhSocket[1], 
	bExecute:= arCloseExecute[1], 
	tTimeout:= T#1S, 
	bBusy=>  arCloseBusy[1], 
	bError=> arCloseError[1], 
	nErrId=> arCloseErrId[1]);



	
CASE iSocket[1] OF 
0:  
    MEMSET(destAddr:= ADR(arhSocket[1]), fillByte:= 0, n:= SIZEOF(arhSocket[1]));  
	arConnectExecute[1]:=FALSE;	
    iSocket[1]:=1;
	
1:  
	iSocket[1]:=2;
		
2:
    arConnectExecute[1]:=TRUE;	
    IF arConnectBusy[1] THEN
	   arConnectExecute[1]:=FALSE;	
       iSocket[1]:=3;
	END_IF	
	
3:  
	iSocket[1]:=4;
	
4:	
    IF arhSocket[1].handle<>0 THEN
       iSocket[1]:=10;
	ELSE IF arConnectError[1] THEN
		    iSocket[1]:=0;
		 END_IF
	END_IF


	   
10:
    arReceiveExecute[1]:=TRUE;
	iSocket[1]:=11;
	
11:
	   arReceiveExecute[1]:=FALSE;
	   iSocket[1]:=12;
12:
	IF NOT arReceiveError[1] AND NOT arReceiveBusy[1] THEN
	   iSocket[1]:=13;
	   ELSE IF arReceiveError[1] THEN
	           iSocket[1]:=90; 
            END_IF  
	END_IF 	
	
13:	
	   iSocket[1]:=20;
	
20:
	arSendExecute[1]:=TRUE; 
	iSocket[1]:=21;


21:	 
	   arSendExecute[1]:=FALSE;
	   iSocket[1]:=22;
	
22:
	IF NOT arSendError[1] AND NOT arSendBusy[1]  THEN
	   iSocket[1]:=23;
	   ELSE IF arSendError[1] THEN
	           iSocket[1]:=90;
	        END_IF
	END_IF 
       		   
23:
	   iSocket[1]:=10;


90: 
    arConnectExecute[1]:=FALSE;  
    arSendExecute[1]:=FALSE;
    arReceiveExecute[1]:=FALSE;
	arCloseExecute[1]:=TRUE;
	iSocket[1]:=91;

91: 
	   iSocket[1]:=92;

92:
	   arCloseExecute[1]:=FALSE;
	   iSocket[1]:=0;

END_CASE
*)
END_ACTION

ACTION TCP2_Server:
tonFS(IN:= TRUE, PT:= T#60S, Q=> , ET=> );

arSocketListen[2](
	sSrvNetId:= , 
	sLocalHost:= '192.168.1.10', 
	nLocalPort:= 6853, 
	bExecute:= arListen[2] OR tonFS.Q , 
	tTimeout:=, 
	bBusy=> arListenBusy[2], 
	bError=> arListenError[2], 
	nErrId=> , 
	hListener=> arhlistener[2]);
	
	
arSocketAccept[2](
	sSrvNetId:= , 
	hListener:= arhlistener[2], 
	bExecute:= arAccept[2], 
	tTimeout:= , 
	bAccepted=> , 
	bBusy=> arAcceptBusy[2], 
	bError=> arAcceptError[2], 
	nErrId=> , 
	hSocket=> arhSocket[2]);	
	
arSocketReceive[2](
	sSrvNetId:= , 
	hSocket:=  arhSocket[2], 
	cbLen:= 255, 
	pDest:= ADR(wReceiveDataBuffer), 
	bExecute:= arReceiveExecute[2], 
	tTimeout:= T#1S, 
	bBusy=> arReceiveBusy[2], 
	bError=> arReceiveError[2], 
	nErrId=> arReceiveErrId[2], 
	nRecBytes=> );

arSocketSend[2](
	sSrvNetId:= , 
	hSocket:= arhSocket[2], 
	cbLen:=  255, 
	pSrc:= ADR(wSendDataBuffer), 
	bExecute:= arSendExecute[2], 
	tTimeout:= T#1S, 
	bBusy=> arSendBusy[2], 
	bError=> arSendError[2], 
	nErrId=> arSendErrId[2]);	
	
	
arSocketClose[2](
	sSrvNetId:= , 
	hSocket:=  arhSocket[2], 
	bExecute:= arCloseExecute[2], 
	tTimeout:= T#1S, 
	bBusy=>  arCloseBusy[2], 
	bError=> arCloseError[2], 
	nErrId=> arCloseErrId[2]);	
	
	
rViewPrintPos:= arRealAxisAdmin[48].o.ActPos- rPrintPosBuffer;
	
CASE iPPAccept OF 
0:  
    MEMSET(destAddr:= ADR(wReceiveData), fillByte:= 0, n:= SIZEOF(wReceiveData));
    MEMSET(destAddr:= ADR(arhSocket[2]), fillByte:= 0, n:= SIZEOF(arhSocket[2]));  		
    iPPAccept:=1;	
1: 	
    IF arhlistener[2].handle<>0 THEN
       iPPAccept:=2;
	END_IF
2:	
	arTon[2](IN:= TRUE, PT:= T#100MS, Q=> , ET=> );	
	IF arTon[2].Q THEN
	   arTon[2](IN:= FALSE, PT:= T#100MS, Q=> , ET=> );	
	   iPPAccept:=10;
	END_IF
	   
10: arAccept[2]:=TRUE;	
    iPPAccept:=11;
	
11:
	arTon[2](IN:= TRUE, PT:= T#100MS, Q=> , ET=> );	
	IF arTon[2].Q THEN
	   arTon[2](IN:= FALSE, PT:= T#100MS, Q=> , ET=> );	
	   iPPAccept:=12;
	END_IF
	
12:	
    IF arhSocket[2].handle<>0 THEN
       iPPAccept:=20;
	   ELSE 
	   arAccept[2]:=FALSE;
	   iPPAccept:=1;
	END_IF

20:
    HMI_PrinterConnected:=TRUE;
    iPPReceive:=10;
	iPPAccept:=100;


90:  
    
    HMI_PrinterConnected:=FALSE;
	arAccept[2]:=FALSE;
    arSendExecute[2]:=FALSE;
    arReceiveExecute[2]:=FALSE;
	arCloseExecute[2]:=TRUE;
	iPPAccept:=91;

91: 
	arTon[2](IN:= TRUE, PT:= T#100MS, Q=> , ET=> );	
	IF arTon[2].Q THEN
	   arTon[2](IN:= FALSE, PT:= T#100MS, Q=> , ET=> );	
	   iPPAccept:=92;
	END_IF
	
92:
	arCloseExecute[2]:=FALSE;
	iPPAccept:=0;
END_CASE
	
CASE iPPReceive OF
	10: 
	    MEMSET(destAddr:= ADR(wReceiveDataBuffer), fillByte:= 0, n:= SIZEOF(wReceiveDataBuffer));
	    arReceiveExecute[2]:=FALSE;
		iPPReceive:=11;
		
	11:
        arTon[3](IN:= TRUE, PT:= T#100MS, Q=> , ET=> );	
		IF arTon[3].Q THEN
		   arTon[3](IN:= FALSE, PT:= T#100MS, Q=> , ET=> );	
		   iPPReceive:=20;
		END_IF
		
	20:	
	    arReceiveExecute[2]:=TRUE;
		iPPReceive:=21;
		
	21:
        arTon[3](IN:= TRUE, PT:= T#1000MS, Q=> , ET=> );	
		IF arTon[3].Q THEN
		   arTon[3](IN:= FALSE, PT:= T#1000MS, Q=> , ET=> );	
		   iPPReceive:=30;
		END_IF		
		
	30: 
        diReceiveData:=MEMCMP(pBuf1:=ADR(wReceiveDataBuffer) , pBuf2:=ADR(wNullData) , n:=SIZEOF(wNullData));
        IF 	diReceiveData<>0 THEN
		    MEMSET(destAddr:= ADR(wReceiveData), fillByte:= 0, n:= SIZEOF(wReceiveData));
		    wReceiveData:=wReceiveDataBuffer;
			pbyReceiveData[0]:=WORD_TO_BYTE(wReceiveDataBuffer[5]);
			pbyReceiveData[1]:=WORD_TO_BYTE(wReceiveDataBuffer[6]);
			pbyReceiveData[2]:=WORD_TO_BYTE(wReceiveDataBuffer[7]);
			pbyReceiveData[3]:=WORD_TO_BYTE(wReceiveDataBuffer[8]);
			pbyReceiveData[4]:=WORD_TO_BYTE(wReceiveDataBuffer[9]);
			pbyReceiveData[5]:=WORD_TO_BYTE(wReceiveDataBuffer[10]);
			pbyReceiveData[6]:=WORD_TO_BYTE(wReceiveDataBuffer[11]);
			pbyReceiveData[7]:=WORD_TO_BYTE(wReceiveDataBuffer[12]);
			pbyReceiveData[8]:=WORD_TO_BYTE(wReceiveDataBuffer[13]);
			pbyReceiveData[9]:=WORD_TO_BYTE(wReceiveDataBuffer[14]);
			pbyReceiveData[10]:=WORD_TO_BYTE(wReceiveDataBuffer[15]);
			pbyReceiveData[11]:=WORD_TO_BYTE(wReceiveDataBuffer[16]);
			pbyReceiveData[12]:=WORD_TO_BYTE(wReceiveDataBuffer[17]);
			pbyReceiveData[13]:=WORD_TO_BYTE(wReceiveDataBuffer[18]);
			pbyReceiveData[14]:=WORD_TO_BYTE(wReceiveDataBuffer[19]);
			pbyReceiveData[15]:=WORD_TO_BYTE(wReceiveDataBuffer[20]);
			pbyReceiveData[16]:=WORD_TO_BYTE(wReceiveDataBuffer[21]);
			pbyReceiveData[17]:=WORD_TO_BYTE(wReceiveDataBuffer[22]);
			pbyReceiveData[18]:=WORD_TO_BYTE(wReceiveDataBuffer[23]);
			pbyReceiveData[19]:=WORD_TO_BYTE(wReceiveDataBuffer[24]);
			pbyReceiveData[20]:=WORD_TO_BYTE(wReceiveDataBuffer[25]);
			pbyReceiveData[21]:=WORD_TO_BYTE(wReceiveDataBuffer[26]);
			pbyReceiveData[22]:=WORD_TO_BYTE(wReceiveDataBuffer[27]);			
	    END_IF
		iPPReceive:=10;
	    IF arSocketReceive[2].bError THEN
		   iPPReceive:=0;
		   iPPAccept:=90;
		END_IF
		
END_CASE

CASE iPPSend OF
	0:  IF HMI_PrinterConnected  AND glb_Un02Box.Box[HMI_PrintNo].PrintRequest AND wReceiveData[0]<>0 THEN
		   iPPSend:=10;
		ELSE IF HMI_PrinterConnected AND wReceiveData[0]<>0 AND  HMI_PrinterTest THEN
                iPPSend:=200;
			 END_IF	
	    END_IF
	10:
	   MEMSET(destAddr:= ADR(byPrintUser), fillByte:= 0, n:= SIZEOF(byPrintUser));
	   MEMSET(destAddr:= ADR(wSendDataBuffer), fillByte:= 0, n:= SIZEOF(wSendDataBuffer));
	   MEMSET(destAddr:= ADR(sAutoPrintData), fillByte:= 0, n:= SIZEOF(sAutoPrintData));
	   iLen:=INT_TO_UINT(LEN(glb_Un02Box.Box[HMI_PrintNo].PrintData));
	   MEMCPY(ADR(sAutoPrintData),ADR(glb_Un02Box.Box[HMI_PrintNo].PrintData),ilen);
	   IF NOT bDebugFlag.0 THEN
	   iPPSend:=11;
	   END_IF
	11:
	   byPrintUser:=MAXSTRING_TO_BYTEARR(sAutoPrintData);
	   IF NOT bDebugFlag.1 THEN
	   iPPSend:=20;
       END_IF
	
	   
	20:		
        wSendDataBuffer[0]:= 35;
		iPPSend:=30;
	30: 	
	    wSendCnt:=wSendCnt+1;
	    IF wSendCnt>200 THEN
		   wSendCnt:=1;
		END_IF	
		
		wSendDataBuffer[1]:=0;
		wSendDataBuffer[2]:=wSendCnt;
		wSendDataBuffer[3]:=0;
		wSendDataBuffer[4]:=44;
		wSendDataBuffer[5]:=BYTE_TO_WORD(byPrintUser[0]);
		wSendDataBuffer[6]:=BYTE_TO_WORD(byPrintUser[1]);
		wSendDataBuffer[7]:=BYTE_TO_WORD(byPrintUser[2]);
		wSendDataBuffer[8]:=BYTE_TO_WORD(byPrintUser[3]);
		wSendDataBuffer[9]:=BYTE_TO_WORD(byPrintUser[4]);
		wSendDataBuffer[10]:=BYTE_TO_WORD(byPrintUser[5]);
		wSendDataBuffer[11]:=BYTE_TO_WORD(byPrintUser[6]);
		wSendDataBuffer[12]:=BYTE_TO_WORD(byPrintUser[7]);
		wSendDataBuffer[13]:=BYTE_TO_WORD(byPrintUser[8]);
		wSendDataBuffer[14]:=BYTE_TO_WORD(byPrintUser[9]);
		wSendDataBuffer[15]:=BYTE_TO_WORD(byPrintUser[10]);
		wSendDataBuffer[16]:=BYTE_TO_WORD(byPrintUser[11]);
		wSendDataBuffer[17]:=BYTE_TO_WORD(byPrintUser[12]);
		wSendDataBuffer[18]:=BYTE_TO_WORD(byPrintUser[13]);
		wSendDataBuffer[19]:=BYTE_TO_WORD(byPrintUser[14]);
		wSendDataBuffer[20]:=BYTE_TO_WORD(byPrintUser[15]);
		wSendDataBuffer[21]:=BYTE_TO_WORD(byPrintUser[16]);
		wSendDataBuffer[22]:=BYTE_TO_WORD(byPrintUser[17]);
		wSendDataBuffer[23]:=BYTE_TO_WORD(byPrintUser[18]);
		wSendDataBuffer[24]:=BYTE_TO_WORD(byPrintUser[19]);
		wSendDataBuffer[25]:=BYTE_TO_WORD(byPrintUser[20]);
        wSendDataBuffer[26]:=BYTE_TO_WORD(byPrintUser[21]);	
		arSendExecute[2]:=FALSE;		
		iPPSend:=31;
		
		
    31:		
	    arTon[4](IN:= TRUE, PT:= T#100MS, Q=> , ET=> );	
		IF arTon[4].Q THEN
		   arTon[4](IN:= FALSE, PT:= T#100MS, Q=> , ET=> );	
		   iPPSend:=40;
		END_IF	
    40:
        arSendExecute[2]:=TRUE;
		iPPSend:=41;	
    41:
	    arTon[4](IN:= TRUE, PT:= T#10S, Q=> , ET=> );	
		IF arTon[4].Q THEN
		   arTon[4](IN:= FALSE, PT:= T#10S, Q=> , ET=> );	
		   iPPSend:=50;
		END_IF
		
	50:	
	    arTon[4](IN:= TRUE, PT:= DINT_TO_TIME(HMI_PrintMaxTime*1000), Q=> , ET=> );	
	    IF wReceiveData[2]=wSendCnt  THEN
		   arTon[4](IN:= FALSE, PT:= DINT_TO_TIME(HMI_PrintMaxTime*1000), Q=> , ET=> );
		   iPPSend:=60;
		   ELSE IF arTon[4].Q THEN
				   arTon[4](IN:= FALSE, PT:= DINT_TO_TIME(HMI_PrintMaxTime*1000), Q=> , ET=> );
				   iPPSend:=51;
		   END_IF
		END_IF
    51: 
	    HMI_PrinterFault:=TRUE;
	    iPPSend:=52;
	52: IF NOT HMI_PrinterFault THEN
		   iPPSend:=60;
	    END_IF
    60:
	
	    glb_Un02Box.Box[HMI_PrintNo].PrintRequest:= FALSE;
		arSendExecute[2]:=FALSE;
	    iPPSend:=0;	

		
	200: 
		MEMSET(destAddr:= ADR(byPrint), fillByte:= 0, n:= SIZEOF(byPrint));
		MEMSET(destAddr:= ADR(wSendDataBuffer), fillByte:= 0, n:= SIZEOF(wSendDataBuffer));
	    MEMSET(destAddr:= ADR(sTestPrintData), fillByte:= 0, n:= SIZEOF(sTestPrintData));
	    iLen:=INT_TO_UINT(LEN(HMI_PrinterTestData));
	    MEMCPY(ADR(sTestPrintData),ADR(HMI_PrinterTestData),ilen);		
	    byPrint:=MAXSTRING_TO_BYTEARR(sTestPrintData);	
		
		iPPSend:=210;	
		
    210:
		wSendDataBuffer[0]:= 35;
		iPPSend:=220;
		
	220:	
	    wSendCnt:=wSendCnt+1;
	    IF wSendCnt>200 THEN
		   wSendCnt:=1;
		END_IF
	
		wSendDataBuffer[1]:=0;
		wSendDataBuffer[2]:=wSendCnt;
		wSendDataBuffer[3]:=0;
		wSendDataBuffer[4]:=44;
		wSendDataBuffer[5]:=BYTE_TO_WORD(byPrint[0]);
		wSendDataBuffer[6]:=BYTE_TO_WORD(byPrint[1]);
		wSendDataBuffer[7]:=BYTE_TO_WORD(byPrint[2]);
		wSendDataBuffer[8]:=BYTE_TO_WORD(byPrint[3]);
		wSendDataBuffer[9]:=BYTE_TO_WORD(byPrint[4]);
		wSendDataBuffer[10]:=BYTE_TO_WORD(byPrint[5]);
		wSendDataBuffer[11]:=BYTE_TO_WORD(byPrint[6]);
		wSendDataBuffer[12]:=BYTE_TO_WORD(byPrint[7]);
		wSendDataBuffer[13]:=BYTE_TO_WORD(byPrint[8]);
		wSendDataBuffer[14]:=BYTE_TO_WORD(byPrint[9]);
		wSendDataBuffer[15]:=BYTE_TO_WORD(byPrint[10]);
		wSendDataBuffer[16]:=BYTE_TO_WORD(byPrint[11]);
		wSendDataBuffer[17]:=BYTE_TO_WORD(byPrint[12]);
		wSendDataBuffer[18]:=BYTE_TO_WORD(byPrint[13]);
		wSendDataBuffer[19]:=BYTE_TO_WORD(byPrint[14]);
		wSendDataBuffer[20]:=BYTE_TO_WORD(byPrint[15]);
		wSendDataBuffer[21]:=BYTE_TO_WORD(byPrint[16]);
		wSendDataBuffer[22]:=BYTE_TO_WORD(byPrint[17]);
		wSendDataBuffer[23]:=BYTE_TO_WORD(byPrint[18]);
		wSendDataBuffer[24]:=BYTE_TO_WORD(byPrint[19]);
		wSendDataBuffer[25]:=BYTE_TO_WORD(byPrint[20]);
        wSendDataBuffer[26]:=BYTE_TO_WORD(byPrint[21]);

		
		arSendExecute[2]:=FALSE;
		iPPSend:=221;
		
    221:		
	    arTon[4](IN:= TRUE, PT:= T#1000MS, Q=> , ET=> );	
		IF arTon[4].Q THEN
		   arTon[4](IN:= FALSE, PT:= T#1000MS, Q=> , ET=> );	
		   iPPSend:=230;
		END_IF	
    230:
        arSendExecute[2]:=TRUE;
		iPPSend:=231;			

    231:
	    arTon[4](IN:= TRUE, PT:= T#1000MS, Q=> , ET=> );	
		IF arTon[4].Q THEN
		   arTon[4](IN:= FALSE, PT:= T#1000MS, Q=> , ET=> );	
		   iPPSend:=240;
		END_IF
		
	240:
	    arTon[4](IN:= TRUE, PT:= DINT_TO_TIME(HMI_PrintMaxTime*1000), Q=> , ET=> );	
	    IF wReceiveData[2]=wSendCnt  THEN
		   arTon[4](IN:= FALSE, PT:= DINT_TO_TIME(HMI_PrintMaxTime*1000), Q=> , ET=> );
		   iPPSend:=0; 
		   arSendExecute[2]:=FALSE;
		   ELSE IF arTon[4].Q THEN
			    arTon[4](IN:= FALSE, PT:= DINT_TO_TIME(HMI_PrintMaxTime*1000), Q=> , ET=> );
				iPPSend:=241;
		   END_IF	   
		END_IF		
		
		
	241: HMI_PrinterFault:=TRUE;
	     arSendExecute[2]:=FALSE;
         iPPSend:=0;	
		
END_CASE
END_ACTION

END_PROGRAM

// ---- Add-On-Instructions/BLINK.TcPOU
FUNCTION_BLOCK BLINK 
VAR_INPUT
	TimeH: DINT;
	TimeL: DINT;
END_VAR
VAR_OUTPUT
	OUT: BOOL;
END_VAR
VAR
	tonTimeHigh: TON;
	tonTimeLow: TON;
END_VAR

tonTimeLow(IN:= NOT tonTimeHigh.Q , PT:=DINT_TO_TIME(TimeL) , Q=> OUT, ET=> );
tonTimeHigh(IN:=tonTimeLow.Q  , PT:= DINT_TO_TIME(TimeH), Q=> , ET=> );

END_FUNCTION_BLOCK

// ---- POUs/IO/IO_Mapping.TcPOU
PROGRAM IO_Mapping
VAR
	i: INT;
	rtsensor: R_trig;
END_VAR

CP02();CP03();CP04();CP05();CP07();CPX1();WPI1();WPI2();

ACTION CP02:
{region "CP02柜"}									
DI_[1,1](	ON:= , 	OFF:= , 	LINK:=EL1008[1,1] , 	VALUE=> 	arDropCylinder[1].i.InSensor	);	(*	料仓1气缸原位	*)
DI_[1,2](	ON:= , 	OFF:= , 	LINK:=EL1008[1,2] , 	VALUE=> 	arDropCylinder[1].i.OutSensor	);	(*	料仓1气缸工作位	*)
DI_[1,3](	ON:= , 	OFF:= , 	LINK:=EL1008[1,3] , 	VALUE=> 	arHighSensor[1].i.Link	);	(*	料仓1少料	*)
DI_[1,4](	ON:= , 	OFF:= , 	LINK:=EL1008[1,4] , 	VALUE=> 	arLowSensor[1].i.Link	);	(*	料仓1缺料	*)
DI_[1,5](	ON:= , 	OFF:= , 	LINK:=EL1008[1,5] , 	VALUE=> 	arDropCylinder[2].i.InSensor	);	(*	料仓2气缸原位	*)
DI_[1,6](	ON:= , 	OFF:= , 	LINK:=EL1008[1,6] , 	VALUE=> 	arDropCylinder[2].i.OutSensor	);	(*	料仓2气缸工作位	*)
DI_[1,7](	ON:= , 	OFF:= , 	LINK:=EL1008[1,7] , 	VALUE=> 	arHighSensor[2].i.Link	);	(*	料仓2少料	*)
DI_[1,8](	ON:= , 	OFF:= , 	LINK:=EL1008[1,8] , 	VALUE=> 	arLowSensor[2].i.Link	);	(*	料仓2缺料	*)
DI_[2,1](	ON:= , 	OFF:= , 	LINK:=EL1008[2,1] , 	VALUE=> 	arDropCylinder[3].i.InSensor	);	(*	料仓3气缸原位	*)
DI_[2,2](	ON:= , 	OFF:= , 	LINK:=EL1008[2,2] , 	VALUE=> 	arDropCylinder[3].i.OutSensor	);	(*	料仓3气缸工作位	*)
DI_[2,3](	ON:= , 	OFF:= , 	LINK:=EL1008[2,3] , 	VALUE=> 	arHighSensor[3].i.Link	);	(*	料仓3少料	*)
DI_[2,4](	ON:= , 	OFF:= , 	LINK:=EL1008[2,4] , 	VALUE=> 	arLowSensor[3].i.Link	);	(*	料仓3缺料	*)
DI_[2,5](	ON:= , 	OFF:= , 	LINK:=EL1008[2,5] , 	VALUE=> 	arDropCylinder[4].i.InSensor	);	(*	料仓4气缸原位	*)
DI_[2,6](	ON:= , 	OFF:= , 	LINK:=EL1008[2,6] , 	VALUE=> 	arDropCylinder[4].i.OutSensor	);	(*	料仓4气缸工作位	*)
DI_[2,7](	ON:= , 	OFF:= , 	LINK:=EL1008[2,7] , 	VALUE=> 	arHighSensor[4].i.Link	);	(*	料仓4少料	*)
DI_[2,8](	ON:= , 	OFF:= , 	LINK:=EL1008[2,8] , 	VALUE=> 	arLowSensor[4].i.Link	);	(*	料仓4缺料	*)
DI_[3,1](	ON:= , 	OFF:= , 	LINK:=EL1008[3,1] , 	VALUE=> 	arDropCylinder[5].i.InSensor	);	(*	料仓5气缸原位	*)
DI_[3,2](	ON:= , 	OFF:= , 	LINK:=EL1008[3,2] , 	VALUE=> 	arDropCylinder[5].i.OutSensor	);	(*	料仓5气缸工作位	*)
DI_[3,3](	ON:= , 	OFF:= , 	LINK:=EL1008[3,3] , 	VALUE=> 	arHighSensor[5].i.Link	);	(*	料仓5少料	*)
DI_[3,4](	ON:= , 	OFF:= , 	LINK:=EL1008[3,4] , 	VALUE=> 	arLowSensor[5].i.Link	);	(*	料仓5缺料	*)
DI_[3,5](	ON:= , 	OFF:= , 	LINK:=EL1008[3,5] , 	VALUE=> 	arDropCylinder[6].i.InSensor	);	(*	料仓6气缸原位	*)
DI_[3,6](	ON:= , 	OFF:= , 	LINK:=EL1008[3,6] , 	VALUE=> 	arDropCylinder[6].i.OutSensor	);	(*	料仓6气缸工作位	*)
DI_[3,7](	ON:= , 	OFF:= , 	LINK:=EL1008[3,7] , 	VALUE=> 	arHighSensor[6].i.Link	);	(*	料仓6少料	*)
DI_[3,8](	ON:= , 	OFF:= , 	LINK:=EL1008[3,8] , 	VALUE=> 	arLowSensor[6].i.Link	);	(*	料仓6缺料	*)
DI_[4,1](	ON:= , 	OFF:= , 	LINK:=EL1008[4,1] , 	VALUE=> 	arDropCylinder[7].i.InSensor	);	(*	料仓7气缸原位	*)
DI_[4,2](	ON:= , 	OFF:= , 	LINK:=EL1008[4,2] , 	VALUE=> 	arDropCylinder[7].i.OutSensor	);	(*	料仓7气缸工作位	*)
DI_[4,3](	ON:= , 	OFF:= , 	LINK:=EL1008[4,3] , 	VALUE=> 	arHighSensor[7].i.Link	);	(*	料仓7少料	*)
DI_[4,4](	ON:= , 	OFF:= , 	LINK:=EL1008[4,4] , 	VALUE=> 	arLowSensor[7].i.Link	);	(*	料仓7缺料	*)
DI_[4,5](	ON:= , 	OFF:= , 	LINK:=EL1008[4,5] , 	VALUE=> 	arDropCylinder[8].i.InSensor	);	(*	料仓8气缸原位	*)
DI_[4,6](	ON:= , 	OFF:= , 	LINK:=EL1008[4,6] , 	VALUE=> 	arDropCylinder[8].i.OutSensor	);	(*	料仓8气缸工作位	*)
DI_[4,7](	ON:= , 	OFF:= , 	LINK:=EL1008[4,7] , 	VALUE=> 	arHighSensor[8].i.Link	);	(*	料仓8少料	*)
DI_[4,8](	ON:= , 	OFF:= , 	LINK:=EL1008[4,8] , 	VALUE=> 	arLowSensor[8].i.Link	);	(*	料仓8缺料	*)
DI_[5,1](	ON:= , 	OFF:= , 	LINK:=EL1008[5,1] , 	VALUE=> 	arDropCylinder[9].i.InSensor	);	(*	料仓9气缸原位	*)
DI_[5,2](	ON:= , 	OFF:= , 	LINK:=EL1008[5,2] , 	VALUE=> 	arDropCylinder[9].i.OutSensor	);	(*	料仓9气缸工作位	*)
DI_[5,3](	ON:= , 	OFF:= , 	LINK:=EL1008[5,3] , 	VALUE=> 	arHighSensor[9].i.Link	);	(*	料仓9少料	*)
DI_[5,4](	ON:= , 	OFF:= , 	LINK:=EL1008[5,4] , 	VALUE=> 	arLowSensor[9].i.Link	);	(*	料仓9缺料	*)
DI_[5,5](	ON:= , 	OFF:= , 	LINK:=EL1008[5,5] , 	VALUE=> 	arDropCylinder[10].i.InSensor	);	(*	料仓10气缸原位	*)
DI_[5,6](	ON:= , 	OFF:= , 	LINK:=EL1008[5,6] , 	VALUE=> 	arDropCylinder[10].i.OutSensor	);	(*	料仓10气缸工作位	*)
DI_[5,7](	ON:= , 	OFF:= , 	LINK:=EL1008[5,7] , 	VALUE=> 	arHighSensor[10].i.Link	);	(*	料仓10少料	*)
DI_[5,8](	ON:= , 	OFF:= , 	LINK:=EL1008[5,8] , 	VALUE=> 	arLowSensor[10].i.Link	);	(*	料仓10缺料	*)
DI_[6,1](	ON:= , 	OFF:= , 	LINK:=EL1008[6,1] , 	VALUE=> 	arDropSensor[1].i.Link	);	(*	工位1落料	*)
DI_[6,2](	ON:= , 	OFF:= , 	LINK:=EL1008[6,2] , 	VALUE=> 	arDropSensor[2].i.Link	);	(*	工位2落料	*)
DI_[6,3](	ON:= , 	OFF:= , 	LINK:=EL1008[6,3] , 	VALUE=> 	arDropSensor[3].i.Link	);	(*	工位3落料	*)
DI_[6,4](	ON:= , 	OFF:= , 	LINK:=EL1008[6,4] , 	VALUE=> 	arDropSensor[4].i.Link	);	(*	工位4落料	*)
DI_[6,5](	ON:= , 	OFF:= , 	LINK:=EL1008[6,5] , 	VALUE=> 	arDropSensor[5].i.Link	);	(*	工位5落料	*)
DI_[6,6](	ON:= , 	OFF:= , 	LINK:=EL1008[6,6] , 	VALUE=> 	arDropSensor[6].i.Link	);	(*	工位6落料	*)
DI_[6,7](	ON:= , 	OFF:= , 	LINK:=EL1008[6,7] , 	VALUE=> 	arDropSensor[7].i.Link	);	(*	工位7落料	*)
DI_[6,8](	ON:= , 	OFF:= , 	LINK:=EL1008[6,8] , 	VALUE=> 	arDropSensor[8].i.Link	);	(*	工位8落料	*)
DI_[7,1](	ON:= , 	OFF:= , 	LINK:=EL1008[7,1] , 	VALUE=> 	arDropSensor[9].i.Link	);	(*	工位9落料	*)
DI_[7,2](	ON:= , 	OFF:= , 	LINK:=EL1008[7,2] , 	VALUE=> 	arDropSensor[10].i.Link	);	(*	工位10落料	*)
DI_[7,3](	ON:= , 	OFF:= , 	LINK:=EL1008[7,3] , 	VALUE=> 	glb_arSafeRelayNo_UN01[1]	);	(*	安全继电器1反馈	*)
DI_[7,4](	ON:= , 	OFF:= , 	LINK:=EL1008[7,4] , 	VALUE=> 	arSafeDoorSts[1]	);	(*	安全门1	*)
DI_[7,5](	ON:= , 	OFF:= , 	LINK:=EL1008[7,5] , 	VALUE=> 	arSafeDoorSts[2]	);	(*	安全门2	*)
DI_[7,6](	ON:= , 	OFF:= , 	LINK:=EL1008[7,6] , 	VALUE=> 	arSafeDoorSts[3]	);	(*	安全门3	*)
DI_[7,7](	ON:= , 	OFF:= , 	LINK:=EL1008[7,7] , 	VALUE=> 	arSafeDoorSts[3]	);	(*	安全门4	*)
DI_[7,8](	ON:= , 	OFF:= , 	LINK:=EL1008[7,8] , 	VALUE=> 	 	);	(*	预留急停反馈	*)
DI_[29,1](	ON:= , 	OFF:= , 	LINK:=EL1008[29,1] , 	VALUE=> 	arRealAxisAdmin[41].i.HomeCali	);	(*	皮带1伺服原点	*)
DI_[29,2](	ON:= , 	OFF:= , 	LINK:=EL1008[29,2] , 	VALUE=> 		);	(*		*)
DI_[29,3](	ON:= , 	OFF:= , 	LINK:=EL1008[29,3] , 	VALUE=> 		);	(*		*)
DI_[29,4](	ON:= , 	OFF:= , 	LINK:=EL1008[29,4] , 	VALUE=> 		);	(*		*)
DI_[29,5](	ON:= , 	OFF:= , 	LINK:=EL1008[29,5] , 	VALUE=> 		);	(*		*)
DI_[29,6](	ON:= , 	OFF:= , 	LINK:=EL1008[29,6] , 	VALUE=> 		);	(*		*)
DI_[29,7](	ON:= , 	OFF:= , 	LINK:=EL1008[29,7] , 	VALUE=> 		);	(*		*)
DI_[29,8](	ON:= , 	OFF:= , 	LINK:=EL1008[29,8] , 	VALUE=> 		);	(*		*)

(*****************************************************************************************************)									
DO_[1,1](	ON:= , 	OFF:= , 	LINK=>EL2008[1,1] , 	VALUE:= 	arDropCylinder[1].o.ValveIn	);	(*	料仓1气缸原位	*)
DO_[1,2](	ON:= , 	OFF:= , 	LINK=>EL2008[1,2] , 	VALUE:= 	arDropCylinder[1].o.ValveOut	);	(*	料仓1气缸工作位	*)
DO_[1,3](	ON:= , 	OFF:= , 	LINK=>EL2008[1,3] , 	VALUE:= 	arDropCylinder[2].o.ValveIn	);	(*	料仓2气缸原位	*)
DO_[1,4](	ON:= , 	OFF:= , 	LINK=>EL2008[1,4] , 	VALUE:= 	arDropCylinder[2].o.ValveOut	);	(*	料仓2气缸工作位	*)
DO_[1,5](	ON:= , 	OFF:= , 	LINK=>EL2008[1,5] , 	VALUE:= 	arDropCylinder[3].o.ValveIn	);	(*	料仓3气缸原位	*)
DO_[1,6](	ON:= , 	OFF:= , 	LINK=>EL2008[1,6] , 	VALUE:= 	arDropCylinder[3].o.ValveOut	);	(*	料仓3气缸工作位	*)
DO_[1,7](	ON:= , 	OFF:= , 	LINK=>EL2008[1,7] , 	VALUE:= 	arDropCylinder[4].o.ValveIn	);	(*	料仓4气缸原位	*)
DO_[1,8](	ON:= , 	OFF:= , 	LINK=>EL2008[1,8] , 	VALUE:= 	arDropCylinder[4].o.ValveOut	);	(*	料仓4气缸工作位	*)
DO_[2,1](	ON:= , 	OFF:= , 	LINK=>EL2008[2,1] , 	VALUE:= 	arDropCylinder[5].o.ValveIn	);	(*	料仓5气缸原位	*)
DO_[2,2](	ON:= , 	OFF:= , 	LINK=>EL2008[2,2] , 	VALUE:= 	arDropCylinder[5].o.ValveOut	);	(*	料仓5气缸工作位	*)
DO_[2,3](	ON:= , 	OFF:= , 	LINK=>EL2008[2,3] , 	VALUE:= 	arDropCylinder[6].o.ValveIn	);	(*	料仓6气缸原位	*)
DO_[2,4](	ON:= , 	OFF:= , 	LINK=>EL2008[2,4] , 	VALUE:= 	arDropCylinder[6].o.ValveOut	);	(*	料仓6气缸工作位	*)
DO_[2,5](	ON:= , 	OFF:= , 	LINK=>EL2008[2,5] , 	VALUE:= 	arDropCylinder[7].o.ValveIn	);	(*	料仓7气缸原位	*)
DO_[2,6](	ON:= , 	OFF:= , 	LINK=>EL2008[2,6] , 	VALUE:= 	arDropCylinder[7].o.ValveOut	);	(*	料仓7气缸工作位	*)
DO_[2,7](	ON:= , 	OFF:= , 	LINK=>EL2008[2,7] , 	VALUE:= 	arDropCylinder[8].o.ValveIn	);	(*	料仓8气缸原位	*)
DO_[2,8](	ON:= , 	OFF:= , 	LINK=>EL2008[2,8] , 	VALUE:= 	arDropCylinder[8].o.ValveOut	);	(*	料仓8气缸工作位	*)
DO_[3,1](	ON:= , 	OFF:= , 	LINK=>EL2008[3,1] , 	VALUE:= 	arDropCylinder[9].o.ValveIn	);	(*	料仓9气缸原位	*)
DO_[3,2](	ON:= , 	OFF:= , 	LINK=>EL2008[3,2] , 	VALUE:= 	arDropCylinder[9].o.ValveOut	);	(*	料仓9气缸工作位	*)
DO_[3,3](	ON:= , 	OFF:= , 	LINK=>EL2008[3,3] , 	VALUE:= 	arDropCylinder[10].o.ValveIn	);	(*	料仓10气缸原位	*)
DO_[3,4](	ON:= , 	OFF:= , 	LINK=>EL2008[3,4] , 	VALUE:= 	arDropCylinder[10].o.ValveOut	);	(*	料仓10气缸工作位	*)
DO_[3,5](	ON:= , 	OFF:= , 	LINK=>EL2008[3,5] , 	VALUE:=     arCounters[1].LineVibrator_Wrk	);	(*	料仓1直震启动	*)
DO_[3,6](	ON:= , 	OFF:= , 	LINK=>EL2008[3,6] , 	VALUE:= 	arCounters[1].CircleVibrator_Wrk	);	(*	料仓1圆震启动	*)
DO_[3,7](	ON:= , 	OFF:= , 	LINK=>EL2008[3,7] , 	VALUE:= 	arCounters[1].DropVibrator_Wrk	);	(*	料仓1落料启动	*)
DO_[3,8](	ON:= , 	OFF:= , 	LINK=>EL2008[3,8] , 	VALUE:= 	arCounters[2].LineVibrator_Wrk	);	(*	料仓2直震启动	*)
DO_[4,1](	ON:= , 	OFF:= , 	LINK=>EL2008[4,1] , 	VALUE:= 	arCounters[2].CircleVibrator_Wrk	);	(*	料仓2圆震启动	*)
DO_[4,2](	ON:= , 	OFF:= , 	LINK=>EL2008[4,2] , 	VALUE:= 	arCounters[2].DropVibrator_Wrk	);	(*	料仓2落料启动	*)
DO_[4,3](	ON:= , 	OFF:= , 	LINK=>EL2008[4,3] , 	VALUE:= 	arCounters[3].LineVibrator_Wrk	);	(*	料仓3直震启动	*)
DO_[4,4](	ON:= , 	OFF:= , 	LINK=>EL2008[4,4] , 	VALUE:= 	arCounters[3].CircleVibrator_Wrk	);	(*	料仓3圆震启动	*)
DO_[4,5](	ON:= , 	OFF:= , 	LINK=>EL2008[4,5] , 	VALUE:= 	arCounters[3].DropVibrator_Wrk	);	(*	料仓3落料启动	*)
DO_[4,6](	ON:= , 	OFF:= , 	LINK=>EL2008[4,6] , 	VALUE:= 	arCounters[4].LineVibrator_Wrk	);	(*	料仓4直震启动	*)
DO_[4,7](	ON:= , 	OFF:= , 	LINK=>EL2008[4,7] , 	VALUE:= 	arCounters[4].CircleVibrator_Wrk	);	(*	料仓4圆震启动	*)
DO_[4,8](	ON:= , 	OFF:= , 	LINK=>EL2008[4,8] , 	VALUE:= 	arCounters[4].DropVibrator_Wrk	);	(*	料仓4落料启动	*)
DO_[5,1](	ON:= , 	OFF:= , 	LINK=>EL2008[5,1] , 	VALUE:= 	arCounters[5].LineVibrator_Wrk	);	(*	料仓5直震启动	*)
DO_[5,2](	ON:= , 	OFF:= , 	LINK=>EL2008[5,2] , 	VALUE:= 	arCounters[5].CircleVibrator_Wrk	);	(*	料仓5圆震启动	*)
DO_[5,3](	ON:= , 	OFF:= , 	LINK=>EL2008[5,3] , 	VALUE:= 	arCounters[5].DropVibrator_Wrk	);	(*	料仓5落料启动	*)
DO_[5,4](	ON:= , 	OFF:= , 	LINK=>EL2008[5,4] , 	VALUE:= 	arCounters[6].LineVibrator_Wrk	);	(*	料仓6直震启动	*)
DO_[5,5](	ON:= , 	OFF:= , 	LINK=>EL2008[5,5] , 	VALUE:= 	arCounters[6].CircleVibrator_Wrk	);	(*	料仓6圆震启动	*)
DO_[5,6](	ON:= , 	OFF:= , 	LINK=>EL2008[5,6] , 	VALUE:= 	arCounters[6].DropVibrator_Wrk	);	(*	料仓6落料启动	*)
DO_[5,7](	ON:= , 	OFF:= , 	LINK=>EL2008[5,7] , 	VALUE:= 	arCounters[7].LineVibrator_Wrk	);	(*	料仓7直震启动	*)
DO_[5,8](	ON:= , 	OFF:= , 	LINK=>EL2008[5,8] , 	VALUE:= 	arCounters[7].CircleVibrator_Wrk	);	(*	料仓7圆震启动	*)
DO_[6,1](	ON:= , 	OFF:= , 	LINK=>EL2008[6,1] , 	VALUE:= 	arCounters[7].DropVibrator_Wrk	);	(*	料仓7落料启动	*)
DO_[6,2](	ON:= , 	OFF:= , 	LINK=>EL2008[6,2] , 	VALUE:= 	arCounters[8].LineVibrator_Wrk	);	(*	料仓8直震启动	*)
DO_[6,3](	ON:= , 	OFF:= , 	LINK=>EL2008[6,3] , 	VALUE:= 	arCounters[8].CircleVibrator_Wrk	);	(*	料仓8圆震启动	*)
DO_[6,4](	ON:= , 	OFF:= , 	LINK=>EL2008[6,4] , 	VALUE:= 	arCounters[8].DropVibrator_Wrk	);	(*	料仓8落料启动	*)
DO_[6,5](	ON:= , 	OFF:= , 	LINK=>EL2008[6,5] , 	VALUE:= 	arCounters[9].LineVibrator_Wrk	);	(*	料仓9直震启动	*)
DO_[6,6](	ON:= , 	OFF:= , 	LINK=>EL2008[6,6] , 	VALUE:= 	arCounters[9].CircleVibrator_Wrk	);	(*	料仓9圆震启动	*)
DO_[6,7](	ON:= , 	OFF:= , 	LINK=>EL2008[6,7] , 	VALUE:= 	arCounters[9].DropVibrator_Wrk	);	(*	料仓9落料启动	*)
DO_[6,8](	ON:= , 	OFF:= , 	LINK=>EL2008[6,8] , 	VALUE:= 	arCounters[10].LineVibrator_Wrk	);	(*	料仓10直震启动	*)
DO_[7,1](	ON:= , 	OFF:= , 	LINK=>EL2008[7,1] , 	VALUE:= 	arCounters[10].CircleVibrator_Wrk	);	(*	料仓10圆震启动	*)
DO_[7,2](	ON:= , 	OFF:= , 	LINK=>EL2008[7,2] , 	VALUE:= 	arCounters[10].DropVibrator_Wrk	);	(*	料仓10落料启动	*)
DO_[7,3](	ON:= , 	OFF:= , 	LINK=>EL2008[7,3] , 	VALUE:= 	glb_bSafetyReset	);	(*	安全继电器1复位	*)
DO_[7,4](	ON:= , 	OFF:= , 	LINK=>EL2008[7,4] , 	VALUE:= 	glb_arLightRed_UN01[1]	);	(*	备用	*)
DO_[7,5](	ON:= , 	OFF:= , 	LINK=>EL2008[7,5] , 	VALUE:= 	glb_arLightYellow_UN01[1]	);	(*	备用	*)
DO_[7,6](	ON:= , 	OFF:= , 	LINK=>EL2008[7,6] , 	VALUE:= 	glb_arLightGreen_UN01[1]	);	(*	备用	*)
DO_[7,7](	ON:= , 	OFF:= , 	LINK=>EL2008[7,7] , 	VALUE:= 	glb_arLightAlarm_UN01[1]	);	(*	备用	*)
DO_[7,8](	ON:= , 	OFF:= , 	LINK=>EL2008[7,8] , 	VALUE:= 		);	(*	备用	*)
									
{endregion}
END_ACTION

